// HMI/VISUs/Cryo-Routines/Cool-Down/VISU_HMI_COOL_DOWN
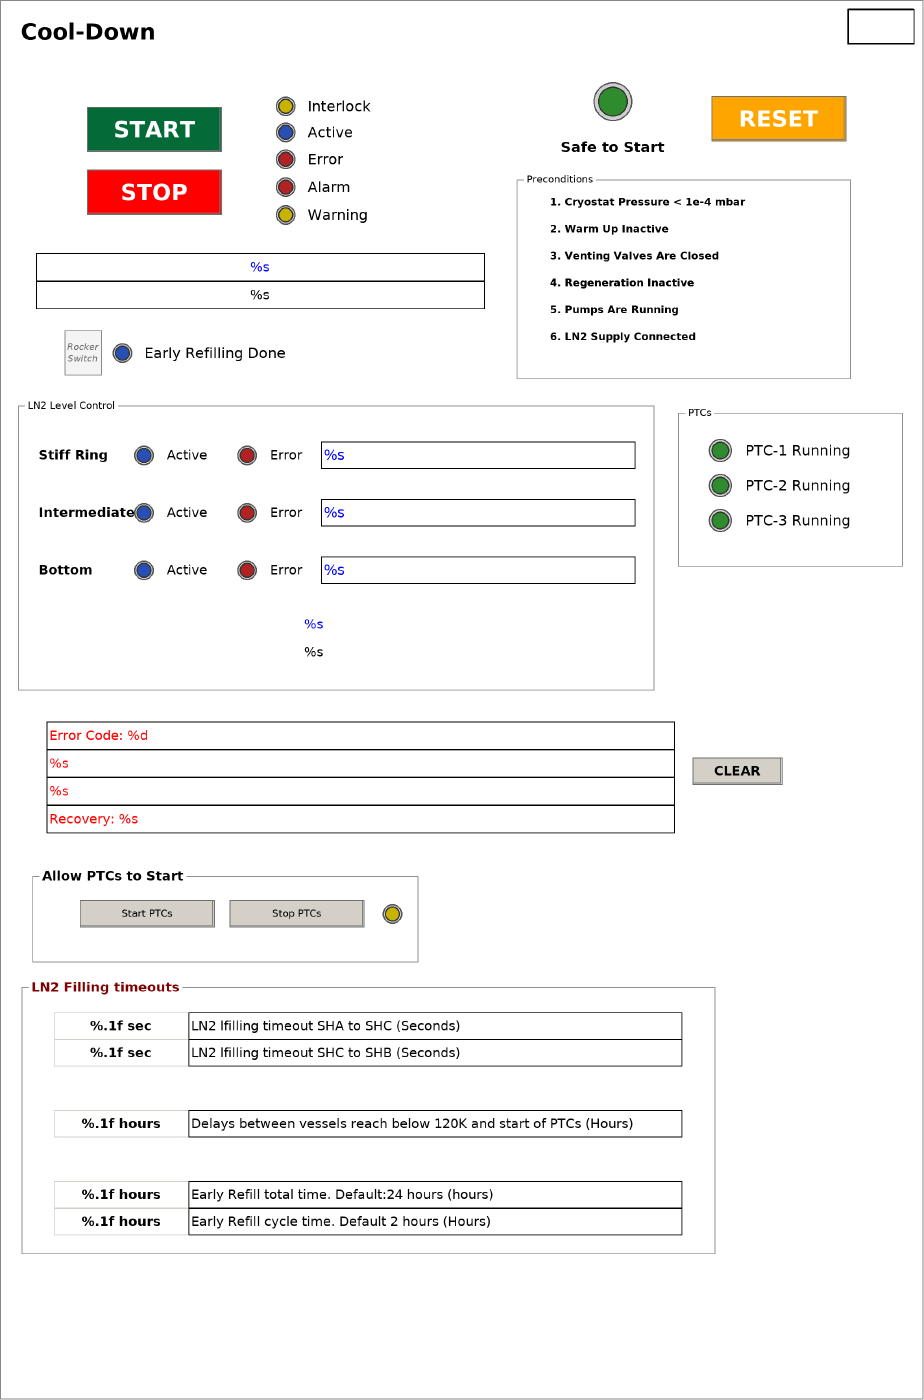
VISUALIZATION VISU_HMI_COOL_DOWN  // 1030x1560
VAR_IN_OUT
	m_instance : FB_METIS_CRYO_COOL_DOWN;
	m_Cry_Instance:	FB_METIS_CRYO_CTRL;	
END_VAR
    Label (20,20 163x30), "Cool-Down"
    Rectangle (40,282 500x31), "%s", text variable: m_instance.stat.sState
    Group (97,103 334x152)
        Group (0,16 150x120)
            Button (0,70 150x50), "STOP"
                OnMouseClick: execute { m_instance.ctrl.bEnable := FALSE; }
            Button (0,0 150x50), "START", input disabled if: NOT m_instance.stat.bPreConditionsMet
                OnMouseClick: execute { m_instance.ctrl.bEnable := TRUE; m_Cry_Instance.ctrl.bEnable_Cool_Down := TRUE; }
        Group (209,0 125x152)
            Label (34,29 91x31), "Active"
            Lamp1 (0,32 25x25), variable: m_instance.stat.bActive, style: Lamp-Lamp1-Blue
            Label (34,59 90x31), "Error"
            Lamp1 (0,62 25x25), variable: m_instance.stat.bError, style: Lamp-Lamp1-Red
            Lamp1 (0,3 25x25), variable: m_instance.interlocks.bInterlock_CoolDown, style: Lamp-Lamp1-Yellow
            Label (34,0 91x31), "Interlock"
            Label (34,90 90x31), "Alarm"
            Lamp1 (0,93 25x25), variable: m_instance.stat.bAlarm, style: Lamp-Lamp1-Red
            Label (34,121 90x31), "Warning"
            Lamp1 (0,124 25x25), variable: m_instance.stat.bWarning, style: Lamp-Lamp1-Yellow
    Lamp1 (658,88 50x50), variable: NOT m_instance.interlocks.bInterlock_CoolDown AND m_instance.stat.bPreConditionsMet, style: Lamp-Lamp1-Green
    Rectangle (608,149 150x30), "Safe to Start"
    GroupBox (576,192 372x230), "Preconditions"
        Rectangle (34,78 300x30), "3. Venting Valves Are Closed", colour toggle: m_instance.in_Cryo_Stat.bVentingValvesAreClosed
        Rectangle (34,108 300x30), "4. Regeneration Inactive", colour toggle: NOT m_instance.in_Cryo_Stat.bRegenerationActive
        Rectangle (34,138 300x30), "5. Pumps Are Running", colour toggle: m_instance.in_Cryo_Stat.bPumpsAreRunning
        Rectangle (34,168 300x30), "6. LN2 Supply Connected", colour toggle: m_instance.bESO_LN2_Supply
    Rectangle (610,300 300x30), "4. Regeneration Inactive", colour toggle: NOT m_instance.in_Cryo_Stat.bRegenerationActive
    Rectangle (610,210 300x30), "1. Cryostat Pressure < 1e-4 mbar", colour toggle: m_instance.in_Cryo_Stat.bInVacuum
    Rectangle (610,240 300x30), "2. Warm Up Inactive", colour toggle: NOT m_instance.in_Cryo_Stat.bWarmUpActive
    Button (793,107 150x50), "RESET", invisible if: NOT m_instance.stat.bError
        OnMouseClick: execute { m_instance.ctrl.bReset := TRUE; }
    Rectangle (52,835 700x31), "%s", text variable: m_instance.stat.Error.sMessage
    Rectangle (52,804 700x31), "Error Code: %d", text variable: m_instance.stat.Error.nCode
    GroupBox (756,452 250x179), "PTCs"
        Group (32,35 187x108)
            Group (0,0 187x30)
                Lamp1 (0,0 30x30), tooltip "If ON, compressor is running", variable: m_Instance.ptc[1].stat.bSystemOn, style: Lamp-Lamp1-Green
                Rectangle (40,0 147x30), "PTC-1 Running", tooltip "Compressor is running"
            Group (0,39 187x30)
                Lamp1 (0,0 30x30), tooltip "If ON, compressor is running", variable: m_Instance.ptc[2].stat.bSystemOn, style: Lamp-Lamp1-Green
                Rectangle (40,0 147x30), "PTC-2 Running", tooltip "Compressor is running"
            Group (0,78 187x30)
                Lamp1 (0,0 30x30), tooltip "If ON, compressor is running", variable: m_Instance.ptc[3].stat.bSystemOn, style: Lamp-Lamp1-Green
                Rectangle (40,0 147x30), "PTC-3 Running", tooltip "Compressor is running"
    GroupBox (20,444 709x325), "LN2 Level Control"
        Group (20,48 668x158)
            Group (0,64 668x30)
                Group (0,0 318x30)
                    Lamp1 (108,3 25x25), tooltip "pump speed > 0 rpm", variable: m_instance.lc_ln2_level_ctrl[2].bActive, style: Lamp-Lamp1-Blue
                    Label (143,0 60x30), "Active"
                    Lamp1 (223,3 25x25), tooltip "pump speed > 0 rpm", variable: m_instance.lc_ln2_level_ctrl[2].bError, style: Lamp-Lamp1-Red
                    Label (258,0 60x30), "Error"
                    Label (0,0 100x30), "Intermediate"
                Rectangle (318,0 350x30), "%s", text variable: m_instance.lc_ln2_level_ctrl[2].LN2_Level.stat.sStatus
            Group (0,128 668x30)
                Group (0,0 318x30)
                    Lamp1 (108,3 25x25), tooltip "pump speed > 0 rpm", variable: m_instance.lc_ln2_level_ctrl[3].bActive, style: Lamp-Lamp1-Blue
                    Label (143,0 60x30), "Active"
                    Lamp1 (223,3 25x25), tooltip "pump speed > 0 rpm", variable: m_instance.lc_ln2_level_ctrl[3].bError, style: Lamp-Lamp1-Red
                    Label (258,0 60x30), "Error"
                    Label (0,0 100x30), "Bottom"
                Rectangle (318,0 350x30), "%s", text variable: m_instance.lc_ln2_level_ctrl[3].LN2_Level.stat.sStatus
            Group (0,0 668x30)
                Group (0,0 318x30)
                    Lamp1 (108,3 25x25), tooltip "pump speed > 0 rpm", variable: m_instance.lc_ln2_level_ctrl[1].bActive, style: Lamp-Lamp1-Blue
                    Label (143,0 60x30), "Active"
                    Lamp1 (223,3 25x25), tooltip "pump speed > 0 rpm", variable: m_instance.lc_ln2_level_ctrl[1].bError, style: Lamp-Lamp1-Red
                    Label (258,0 60x30), "Error"
                    Label (0,0 100x30), "Stiff Ring"
                Rectangle (318,0 350x30), "%s", text variable: m_instance.lc_ln2_level_ctrl[1].LN2_Level.stat.sStatus
        Rectangle (80,236 500x31), "%s", text variable: m_instance.stat.sEarlyFillState
        Rectangle (80,267 500x31), "%s", text variable: m_instance.stat.sEarlyFillSubState
    Rectangle (52,866 700x31), "%s", text variable: m_instance.stat.sErrorMessage
    Rectangle (52,897 700x31), "Recovery: %s", text variable: m_instance.stat.sRecoverySuggestion
    Frame (945,10 75x40)
        shows VISU_HMI_SUBSYSTEM_BUTTON(m_Hmi := PRG_HMI.fbBackButton)
        OnMouseClick: execute { PRG_HMI.eActiveTab := PRG_HMI.ePreviousTab; }
    Rectangle (40,313 500x31), "%s", text variable: m_instance.stat.sSubState
    GroupBox (36,968 430x104), "Allow PTCs to Start"
        Button (53,35 150x30), "Start PTCs", tooltip "Allow PTCs to start"
            OnMouseClick: execute { m_instance.bAllowPTCsStart := TRUE; }
        Button (220,35 150x30), "Stop PTCs", tooltip "Do not allow PTCs to start"
            OnMouseClick: execute { m_instance.bAllowPTCsStart := FALSE; }
        Lamp1 (389,38 25x25), variable: m_instance.bAllowPTCsStart, style: Lamp-Lamp1-Yellow
    GroupBox (24,1092 773x305), "LN2 Filling timeouts"
        Group (36,36 700x248)
            Group (0,0 700x60)
                Group (0,0 700x30)
                    Textfield (0,0 150x30), "%.1f sec", tooltip "(Seconds) LN2 lfilling timeout SHA to SHC", text variable: m_instance.lrDelaySHC
                        OnMouseClick: write the text variable via Default
                    Rectangle (150,0 550x30), "LN2 lfilling timeout SHA to SHC (Seconds)", text variable: m_instance.lrDelaySHC
                Group (0,30 700x30)
                    Textfield (0,0 150x30), "%.1f sec", tooltip "(Seconds) LN2 lfilling timeout SHC to SHB", text variable: m_instance.lrDelaySHB
                        OnMouseClick: write the text variable via Default
                    Rectangle (150,0 550x30), "LN2 lfilling timeout SHC to SHB (Seconds)"
            Group (0,109 700x30)
                Textfield (0,0 150x30), "%.1f hours", tooltip "(Hours) delays between vessels reach below 120K and start of PTCs", text variable: m_instance.lrDelaySHCold
                    OnMouseClick: write the text variable via Default
                Rectangle (150,0 550x30), "Delays between vessels reach below 120K and start of PTCs (Hours)"
            Group (0,188 700x60)
                Group (0,0 700x30)
                    Textfield (0,0 150x30), "%.1f hours", tooltip "(Hours) Early Refill total time (24 hours)", text variable: m_instance.lrEarlyRefillTotal
                        OnMouseClick: write the text variable via Default
                    Rectangle (150,0 550x30), "Early Refill total time. Default:24 hours (hours)"
                Group (0,30 700x30)
                    Textfield (0,0 150x30), "%.1f hours", tooltip "(Hours) Early Refill cycle time.", text variable: m_instance.lrEarlyRefillCycle
                        OnMouseClick: write the text variable via Default
                    Rectangle (150,0 550x30), "Early Refill cycle time. Default 2 hours (Hours)"
    Group (72,368 253x50)
        RockerSwitch (0,0 41x50), variable: m_instance.bEarlyRefillDone, behaviour: TOGGLE, style: Switch-RockerSwitch-Blue
        Lamp1 (52,13 25x25), variable: m_instance.bEarlyRefillDone, style: Lamp-Lamp1-Blue
        Label (86,10 167x31), "Early Refilling Done"
    Button (772,844 100x30), "CLEAR", tooltip "Clears Error texts"
        OnMouseClick: execute {
            m_instance.stat.Error.nCode := 0;
            m_instance.stat.Error.sMessage:= '';
            m_instance.stat.sErrorMessage := '';
            m_instance.stat.sRecoverySuggestion := '';
        }
END_VISUALIZATION

// HMI/VISUs/Cryo-Routines/Evacuation/VISU_HMI_EVACUATION
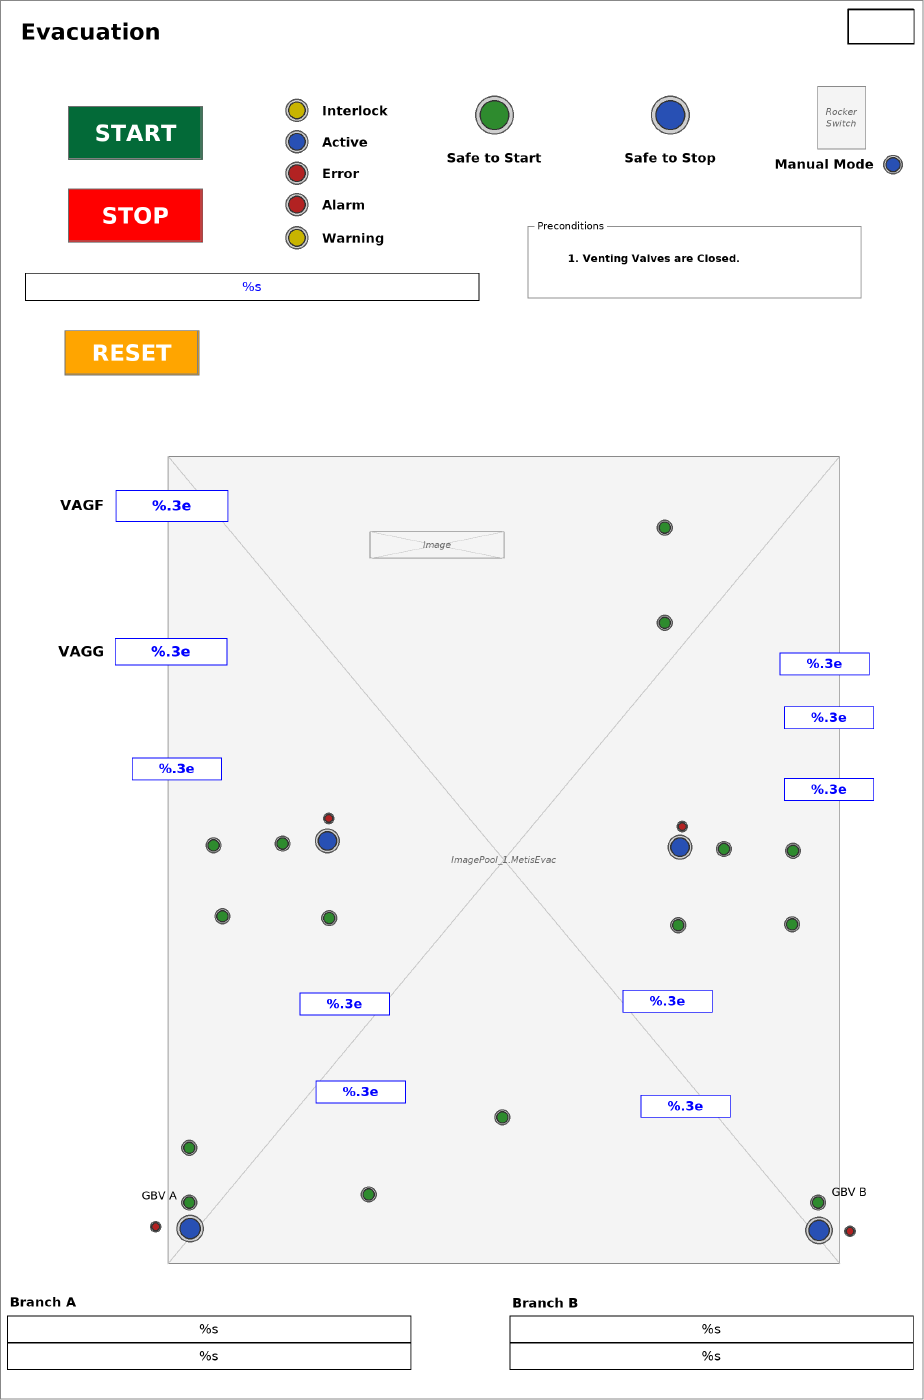
VISUALIZATION VISU_HMI_EVACUATION  // 1030x1560
    Label (20,20 163x30), "Evacuation"
    Frame (0,0 1030x1560)
        shows TEMPLATE_EVACUATION(m_Instance := MAIN.met_cryo_ctrl.met_evac, m_venting_instance := MAIN.met_cryo_ctrl.met_venting, m_cool_down_instance := MAIN.met_cryo_ctrl.met_cool_down)
    Frame (945,10 75x40)
        shows VISU_HMI_SUBSYSTEM_BUTTON(m_Hmi := PRG_HMI.fbBackButton)
        OnMouseClick: execute { PRG_HMI.eActiveTab := PRG_HMI.ePreviousTab; }
END_VISUALIZATION

// HMI/VISUs/Cryo-Routines/Power-Outage/VISU_HMI_POWER_OUTAGE
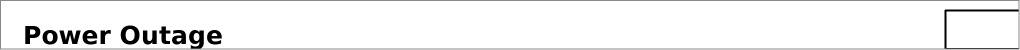
VISUALIZATION VISU_HMI_POWER_OUTAGE  // 1020x50
    Label (20,20 208x30), "Power Outage"
    Frame (945,10 75x40)
        shows VISU_HMI_SUBSYSTEM_BUTTON(m_Hmi := PRG_HMI.fbBackButton)
        OnMouseClick: execute { PRG_HMI.eActiveTab := PRG_HMI.ePreviousTab; }
END_VISUALIZATION

// HMI/VISUs/Cryo-Routines/Regeneration/VISU_HMI_REGENERATION
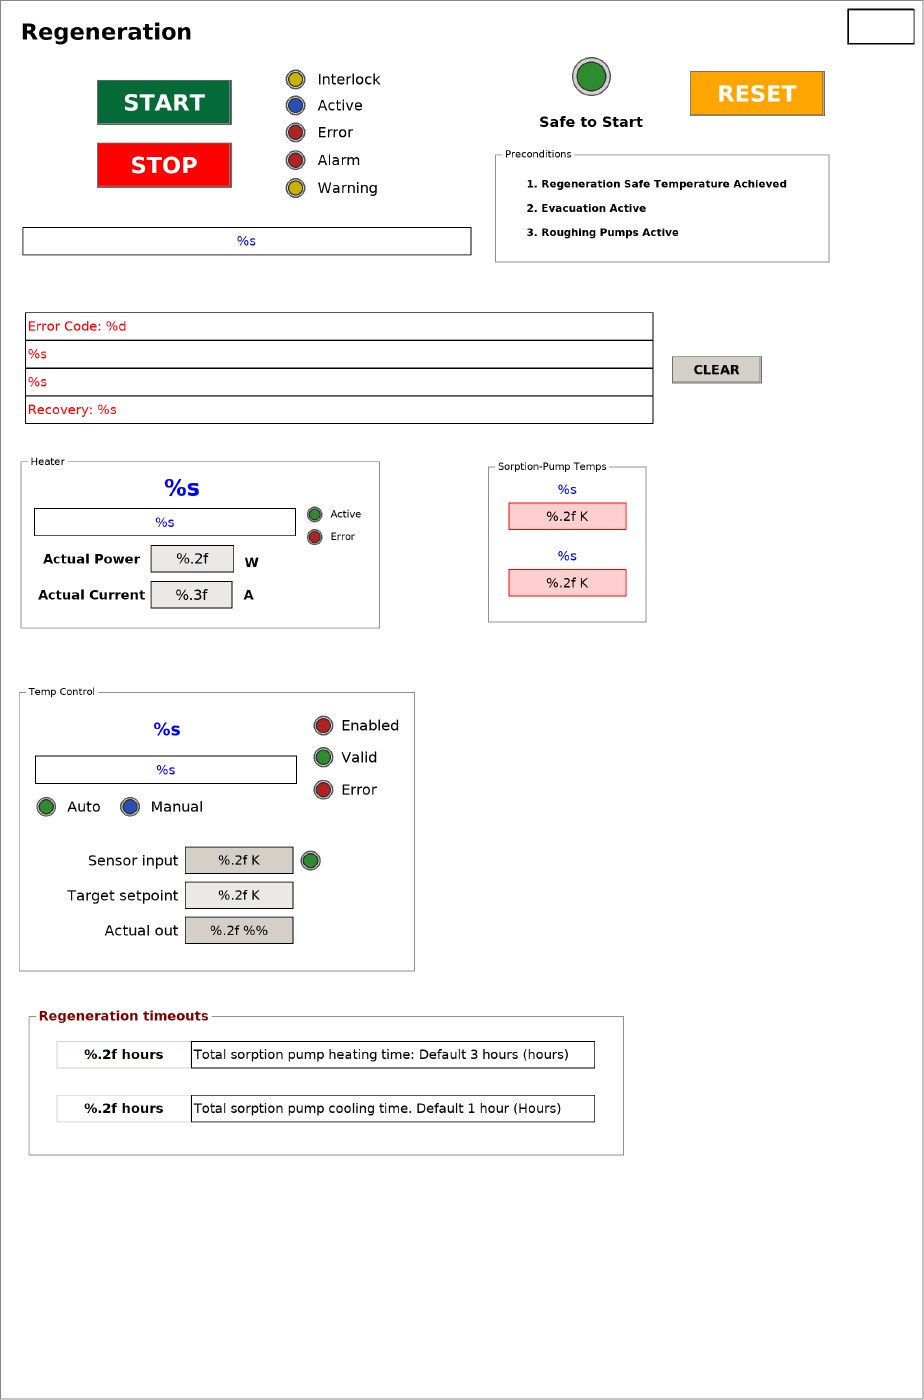
VISUALIZATION VISU_HMI_REGENERATION  // 1030x1560
VAR_IN_OUT
	//m_temp_instance : FB_METIS_TEMPERATURES;
	m_instance : FB_METIS_CRYO_REGENERATION;
	
END_VAR
    Label (20,20 194x30), "Regeneration"
    Frame (12,760 450x322)
        shows TEMPLATE_METIS_CTRL_TEMPERATURE_SIMPLIFIED(m_instance := MAIN.met_cryo_ctrl.met_tctrl.tc_cry_sp)
    Frame (16,504 407x196)
        shows TEMPLATE_METIS_HEATER_SIMPLIFIED(m_instance := MAIN.met_cryo_ctrl.met_heaters.h_cry_sp)
    Group (544,512 176x181)
        GroupBox (0,0 176x181), "Sorption-Pump Temps"
        Group (13,18 150x144)
            Frame (0,0 150x70)
                shows TEMPLATE_TEMP_SENSOR_VALUE_ONLY(m_instance := MAIN.met_cryo_ctrl.met_temp.t_cry_sp_1)
            Frame (0,74 150x70)
                shows TEMPLATE_TEMP_SENSOR_VALUE_ONLY(m_instance := MAIN.met_cryo_ctrl.met_temp.t_cry_sp_2)
    Rectangle (25,253 500x31), "%s", text variable: m_instance.stat.sState
    Group (108,73 334x152)
        Button (0,86 150x50), "STOP"
            OnMouseClick: execute { m_instance.ctrl.bEnable := FALSE; }
        Button (0,16 150x50), "START", input disabled if: m_instance.interlocks.bInterlock_Regeneration OR NOT m_instance.stat.bPreConditionsMet
            OnMouseClick: execute { m_instance.ctrl.bEnable := TRUE; }
        Group (209,0 125x152)
            Label (34,29 91x31), "Active"
            Lamp1 (0,32 25x25), variable: m_instance.stat.bActive, style: Lamp-Lamp1-Blue
            Label (34,59 90x31), "Error"
            Lamp1 (0,62 25x25), variable: m_instance.stat.bError, style: Lamp-Lamp1-Red
            Lamp1 (0,3 25x25), variable: m_instance.interlocks.bInterlock_Regeneration, style: Lamp-Lamp1-Yellow
            Label (34,0 91x31), "Interlock"
            Label (34,90 90x31), "Alarm"
            Lamp1 (0,93 25x25), variable: m_instance.stat.bAlarm, style: Lamp-Lamp1-Red
            Label (34,121 90x31), "Warning"
            Lamp1 (0,124 25x25), variable: m_instance.stat.bWarning, style: Lamp-Lamp1-Yellow
    Lamp1 (634,60 50x50), variable: NOT m_instance.interlocks.bInterlock_Regeneration, style: Lamp-Lamp1-Green
    Rectangle (584,121 150x30), "Safe to Start"
    GroupBox (552,164 372x128), "Preconditions"
        Rectangle (32,80 300x30), "3. Roughing Pumps Active", colour toggle: m_instance.in_Cryo_Stat.bRoughingPumpsAreRunning
    Rectangle (584,190 300x30), "1. Regeneration Safe Temperature Achieved", colour toggle: (m_instance.in_Cryo_Stat.lrLowestTempK >= m_instance.in_lrRegeneration_Safe_Temp)
    Rectangle (584,217 300x30), "2. Evacuation Active", colour toggle: m_instance.in_Cryo_Stat.bEvacuationActive
    Button (769,79 150x50), "RESET", invisible if: NOT m_instance.stat.bError
        OnMouseClick: execute { m_instance.ctrl.bReset := TRUE; }
    Frame (945,10 75x40)
        shows VISU_HMI_SUBSYSTEM_BUTTON(m_Hmi := PRG_HMI.fbBackButton)
        OnMouseClick: execute { PRG_HMI.eActiveTab := PRG_HMI.ePreviousTab; }
    Rectangle (28,379 700x31), "%s", text variable: m_instance.stat.Error.sMessage
    Rectangle (28,348 700x31), "Error Code: %d", text variable: m_instance.stat.Error.nCode
    Rectangle (28,410 700x31), "%s", text variable: m_instance.stat.sErrorMessage
    Rectangle (28,441 700x31), "Recovery: %s", text variable: m_instance.stat.sRecoverySuggestion
    GroupBox (32,1124 663x163), "Regeneration timeouts"
        Group (31,36 600x90)
            Group (0,0 600x30)
                Textfield (0,0 150x30), "%.2f hours", tooltip "(Hours) Total heating time", text variable: m_instance.lrHeatingTime
                    OnMouseClick: write the text variable via Default
                Rectangle (150,0 450x30), "Total sorption pump heating time: Default 3 hours (hours)"
            Group (0,60 600x30)
                Textfield (0,0 150x30), "%.2f hours", tooltip "(Hours) Total Cooling time", text variable: m_instance.lrCoolDownTime
                    OnMouseClick: write the text variable via Default
                Rectangle (150,0 450x30), "Total sorption pump cooling time. Default 1 hour (Hours)"
    Button (749,397 100x30), "CLEAR", tooltip "Clears Error texts"
        OnMouseClick: execute {
            m_instance.stat.Error.nCode := 0;
            m_instance.stat.Error.sMessage:= '';
            m_instance.stat.sErrorMessage := '';
            m_instance.stat.sRecoverySuggestion := '';
        }
END_VISUALIZATION

// HMI/VISUs/Cryo-Routines/Regeneration/VISU_REGENERATION_CTRL
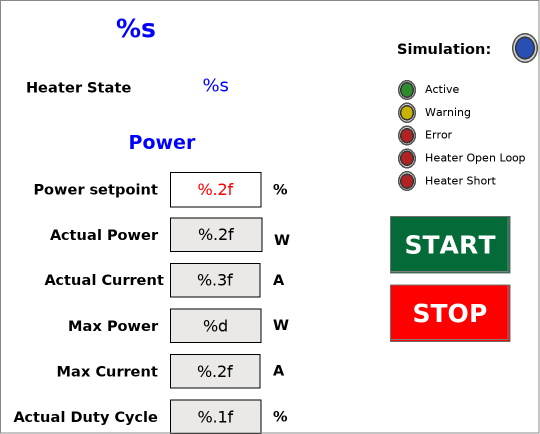
VISUALIZATION VISU_REGENERATION_CTRL  // 540x434
    Frame (0,0 540x434)
        shows TEMPLATE_HEATER_PWM_CTRL(m_instance := MAIN.met_cryo_ctrl.met_regeneration.h_sorption_pump_heater, m_bEnable := MAIN.met_cryo_ctrl.met_regeneration.h_sorption_pump_heater.ctrl.bEnable)
END_VISUALIZATION

// HMI/VISUs/Cryo-Routines/Regeneration/VISU_SORPTION_HEATER
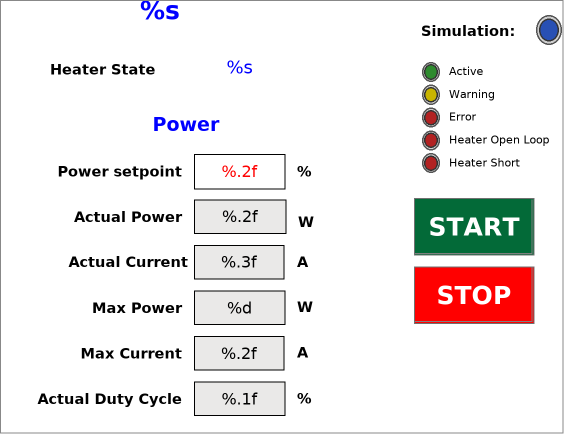
VISUALIZATION VISU_SORPTION_HEATER  // 564x434
    Frame (24,-18 540x434)
        shows TEMPLATE_HEATER_PWM_CTRL(m_instance := MAIN.met_cryo_ctrl.met_regeneration.h_sorption_pump_heater, m_bEnable := MAIN.met_cryo_ctrl.met_regeneration.h_sorption_pump_heater.ctrl.bEnable)
END_VISUALIZATION

// HMI/VISUs/Cryo-Routines/Regeneration/VISU_SORPTION_TEMP_VOTE
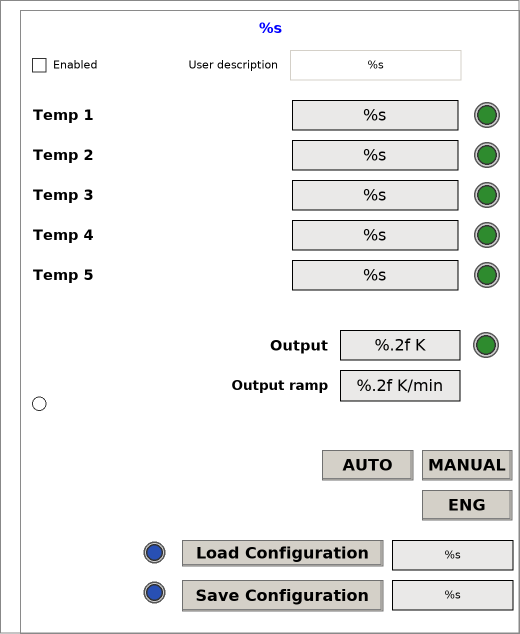
VISUALIZATION VISU_SORPTION_TEMP_VOTE  // 520x634
    Frame (20,10 500x624)
        shows TEMPLATE_TEMPERATURE_VOTE(m_Instance := MAIN.met_cryo_ctrl.met_regeneration.t_vote_tc_cry_sp, m_all_temperatures_array := MAIN.met_cryo_ctrl.met_temp)
END_VISUALIZATION

// HMI/VISUs/Cryo-Routines/Venting/VISU_HMI_VENTING
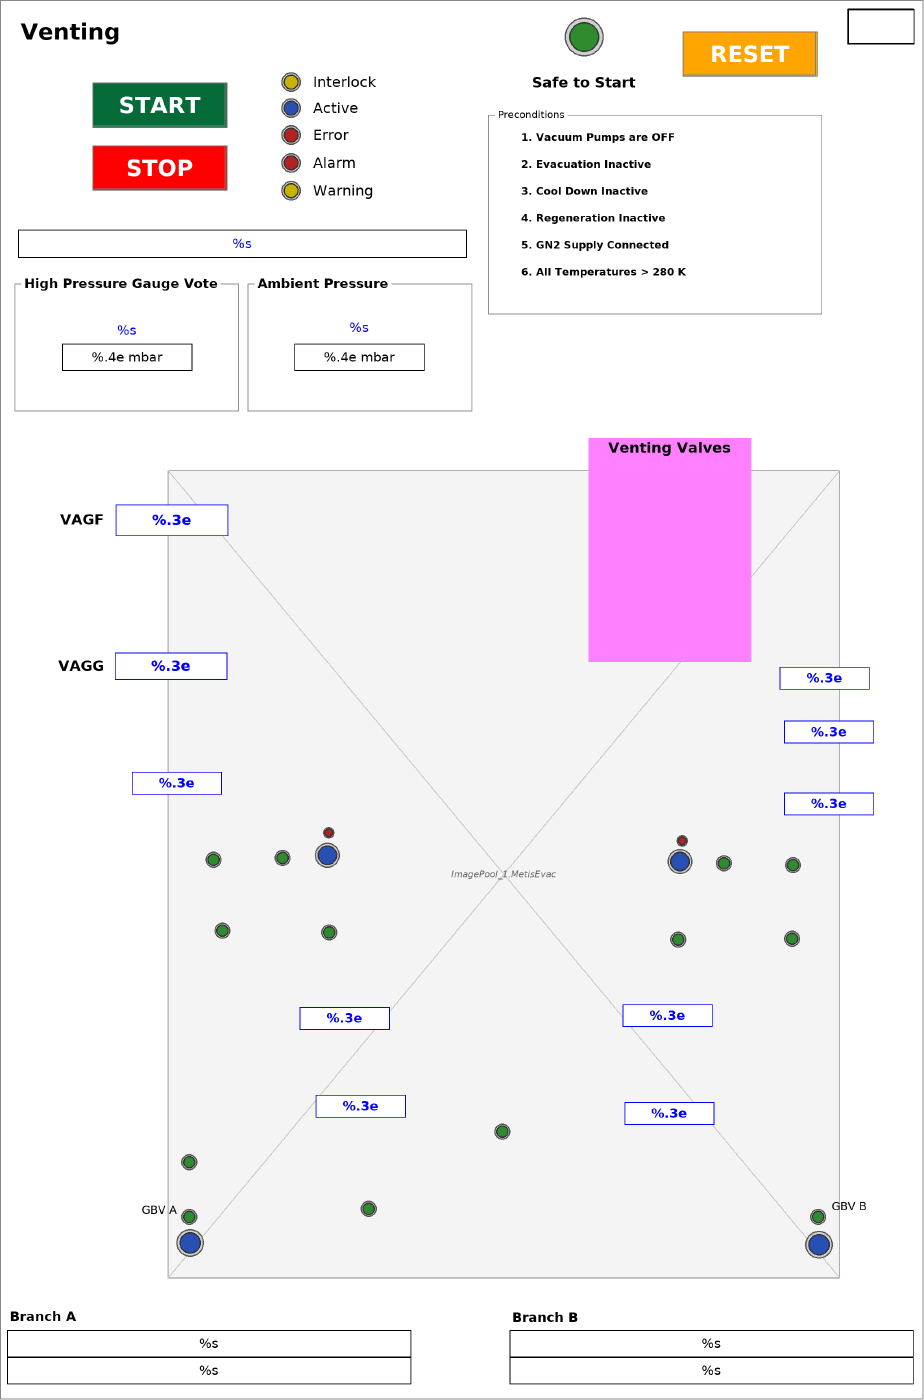
VISUALIZATION VISU_HMI_VENTING  // 1030x1560
VAR_IN_OUT
	m_Instance : FB_METIS_CRYO_VENTING;
	m_Cry_Instance:	FB_METIS_CRYO_CTRL;
END_VAR
    Image (187,524 749x900), image: ImagePool_1.MetisEvac
    Label (20,20 163x30), "Venting"
    Rectangle (20,256 500x31), "%s", text variable: m_instance.stat.sState
    Button (103,162 150x50), "STOP"
        OnMouseClick: execute { m_instance.ctrl.bEnable := FALSE; m_Cry_Instance.ctrl.bEnable_Venting := FALSE; }
    Button (103,92 150x50), "START", input disabled if: NOT m_instance.stat.bPreConditionsMet OR m_instance.interlocks.bInterlock_Venting
        OnMouseClick: execute { m_instance.ctrl.bEnable := TRUE; m_Cry_Instance.ctrl.bEnable_Venting := TRUE; }
    Label (346,105 91x31), "Active"
    Lamp1 (312,108 25x25), variable: m_instance.stat.bActive, style: Lamp-Lamp1-Blue
    Label (346,135 90x31), "Error"
    Lamp1 (312,138 25x25), variable: m_instance.stat.bError, style: Lamp-Lamp1-Red
    Lamp1 (312,79 25x25), variable: m_instance.interlocks.bInterlock_Venting, style: Lamp-Lamp1-Yellow
    Label (346,76 91x31), "Interlock"
    Label (346,166 90x31), "Alarm"
    Lamp1 (312,169 25x25), variable: m_instance.stat.bAlarm, style: Lamp-Lamp1-Red
    Label (346,197 90x31), "Warning"
    Lamp1 (312,200 25x25), variable: m_instance.stat.bWarning, style: Lamp-Lamp1-Yellow
    Lamp1 (626,16 50x50), variable: NOT m_instance.interlocks.bInterlock_Venting AND m_instance.stat.bPreConditionsMet, style: Lamp-Lamp1-Green
    Rectangle (576,77 150x30), "Safe to Start"
    GroupBox (544,120 372x230), "Preconditions"
        Rectangle (34,78 300x30), "3. Cool Down Inactive", colour toggle: NOT m_instance.in_Cryo_Stat.bCoolDownActive
        Rectangle (34,108 300x30), "4. Regeneration Inactive", colour toggle: NOT m_instance.in_Cryo_Stat.bRegenerationActive
        Rectangle (34,138 300x30), "5. GN2 Supply Connected", colour toggle: m_instance.in_Cryo_Stat.bGN2SupplyConnected
        Rectangle (34,168 300x30), "6. All Temperatures > 280 K", colour toggle: m_instance.in_Cryo_Stat.lrLowestTempK > 280.0
    Rectangle (578,138 300x30), "1. Vacuum Pumps are OFF", colour toggle: NOT m_instance.in_Cryo_Stat.bPumpsAreRunning
    Rectangle (578,168 300x30), "2. Evacuation Inactive", colour toggle: NOT m_instance.in_Cryo_Stat.bEvacuationActive
    Button (761,35 150x50), "RESET", invisible if: NOT m_instance.stat.bError
        OnMouseClick: execute { m_instance.ctrl.bReset := TRUE; }
    Frame (945,10 75x40)
        shows VISU_HMI_SUBSYSTEM_BUTTON(m_Hmi := PRG_HMI.fbBackButton)
        OnMouseClick: execute { PRG_HMI.eActiveTab := PRG_HMI.ePreviousTab; }
    GroupBox (276,308 250x150), "Ambient Pressure"
        Frame (50,40 150x70)
            shows TEMPLATE_AMBIENT_PRESSURE_READING(m_instance := MAIN.met_cryo_ctrl.sensor_AMB_PRESS)
    GroupBox (16,308 250x150), "High Pressure Gauge Vote", tooltip "Pressure vote of HPG1 and HPG2"
        Group (53,45 145x60)
            Rectangle (0,30 145x30), "%.4e mbar", tooltip "Pressure in mbar", text variable: m_instance.HPG.stat.lrPressure
            Rectangle (0,0 145x30), "%s", text variable: m_instance.HPG.in_sName
    Rectangle (8,1482 450x30), "%s", text variable: m_Cry_Instance.met_evac.evac_branch_a.stat.sErrorText
    Rectangle (8,1512 450x30), "%s", text variable: m_Cry_Instance.met_evac.evac_branch_a.stat.sStatus
    Rectangle (8,1452 100x30), "Branch A"
    Rectangle (568,1482 450x30), "%s", text variable: m_Cry_Instance.met_evac.evac_branch_b.stat.sErrorText
    Rectangle (568,1512 450x30), "%s", text variable: m_Cry_Instance.met_evac.evac_branch_b.stat.sStatus
    Rectangle (568,1453 100x30), "Branch B"
    Rectangle (334,1122 100x25), "%.3e", text variable: m_Cry_Instance.met_evac.evac_branch_a.VAG1.stat.lrPressure
    Rectangle (147,860 100x25), "%.3e", text variable: m_Cry_Instance.met_evac.evac_branch_a.VAG2.stat.lrPressure
    Lamp1 (194,1367 36x36), variable: m_Cry_Instance.met_evac.evac_branch_a.rp.stat.bReady, style: Lamp-Lamp1-Blue
    Lamp1 (349,937 32x32), tooltip "If ON, TMP pump is at its nominal speed, i.e. Ready.", variable: m_Cry_Instance.met_evac.evac_branch_a.tp.stat.bReady, style: Lamp-Lamp1-Blue
    Lamp1 (238,1027 20x20), variable: m_Cry_Instance.met_evac.evac_branch_a.PVV1.stat.bActON, style: Lamp-Lamp1-Green
    Lamp1 (357,1029 20x20), variable: m_Cry_Instance.met_evac.evac_branch_a.PVV2.stat.bActON, style: Lamp-Lamp1-Green
    Lamp1 (228,948 20x20), variable: m_Cry_Instance.met_evac.evac_branch_a.PVV3.stat.bActON, style: Lamp-Lamp1-Green
    Lamp1 (305,946 20x20), variable: m_Cry_Instance.met_evac.evac_branch_a.PVV4.stat.bActON, style: Lamp-Lamp1-Green
    Lamp1 (201,1346 20x20), variable: m_Cry_Instance.met_evac.evac_branch_a.GBV.stat.bActON, style: Lamp-Lamp1-Green
    Lamp1 (359,921 15x14), tooltip "If ON, TMP pump is still spinning.", variable: m_Cry_Instance.met_evac.evac_branch_a.tp.stat.bSpeed100, style: Lamp-Lamp1-Red
    Rectangle (352,1220 100x25), "%.3e", text variable: m_Cry_Instance.met_evac.evac_branch_a.VAG3.stat.lrPressure
    Lamp1 (742,944 32x32), tooltip "If ON, TMP pump is at its nominal speed, i.e. Ready.", variable: m_Cry_Instance.met_evac.evac_branch_b.tp.stat.bReady, style: Lamp-Lamp1-Blue
    Lamp1 (753,930 15x14), tooltip "If ON, TMP pump is still spinning.", variable: m_Cry_Instance.met_evac.evac_branch_b.tp.stat.bSpeed100, style: Lamp-Lamp1-Red
    Lamp1 (797,952 20x20), variable: m_Cry_Instance.met_evac.evac_branch_b.PVV4.stat.bActON, style: Lamp-Lamp1-Green
    Lamp1 (874,954 20x20), variable: m_Cry_Instance.met_evac.evac_branch_b.PVV3.stat.bActON, style: Lamp-Lamp1-Green
    Lamp1 (746,1037 20x20), variable: m_Cry_Instance.met_evac.evac_branch_b.PVV2.stat.bActON, style: Lamp-Lamp1-Green
    Lamp1 (873,1036 20x20), variable: m_Cry_Instance.met_evac.evac_branch_b.PVV1.stat.bActON, style: Lamp-Lamp1-Green
    Lamp1 (895,1369 36x36), variable: m_Cry_Instance.met_evac.evac_branch_b.rp.stat.bReady, style: Lamp-Lamp1-Blue
    Lamp1 (902,1346 20x20), variable: m_Cry_Instance.met_evac.evac_branch_b.GBV.stat.bActON, style: Lamp-Lamp1-Green
    Rectangle (696,1228 100x25), "%.3e", text variable: m_Cry_Instance.met_evac.evac_branch_b.VAG3.stat.lrPressure
    Rectangle (874,883 100x25), "%.3e", text variable: m_Cry_Instance.met_evac.evac_branch_b.VAG2.stat.lrPressure
    Rectangle (694,1119 100x25), "%.3e", text variable: m_Cry_Instance.met_evac.evac_branch_b.VAG1.stat.lrPressure
    Lamp1 (728,592 25x25), variable: m_Instance.N2V_1.stat.bActON, style: Lamp-Lamp1-Green
    Lamp1 (728,696 25x25), variable: m_Instance.N2V_2.stat.bActON, style: Lamp-Lamp1-Green
    Lamp1 (201,1285 20x20), variable: m_Cry_Instance.met_cool_down.PVV_P1.stat.bActON, style: Lamp-Lamp1-Green
    Lamp1 (401,1337 20x20), variable: m_Cry_Instance.met_cool_down.PVV_P3.stat.bActON, style: Lamp-Lamp1-Green
    Lamp1 (550,1251 20x20), variable: m_Cry_Instance.met_cool_down.PVV_P2.stat.bActON, style: Lamp-Lamp1-Green
    Rectangle (150,1333 55x30), "GBV A"
    Rectangle (919,1329 55x30), "GBV B"
    Rectangle (129,562 125x35), "%.3e", text variable: m_Cry_Instance.met_evac.VAGF.stat.lrPressure
    Rectangle (54,564 75x30), "VAGF"
    Rectangle (128,727 125x30), "%.3e", text variable: m_Cry_Instance.met_evac.VAGG.stat.lrPressure
    Rectangle (53,727 75x30), "VAGG"
    Rectangle (869,743 100x25), "%.3e", text variable: m_Instance.sensor_HPG1.stat.lrPressure
    Rectangle (874,803 100x25), "%.3e", text variable: m_Instance.sensor_HPG2.stat.lrPressure
    Rectangle (656,488 181x249), "Venting Valves"
END_VISUALIZATION

// HMI/VISUs/Cryo-Routines/Warm-Up/VISU_HMI_WARM_UP
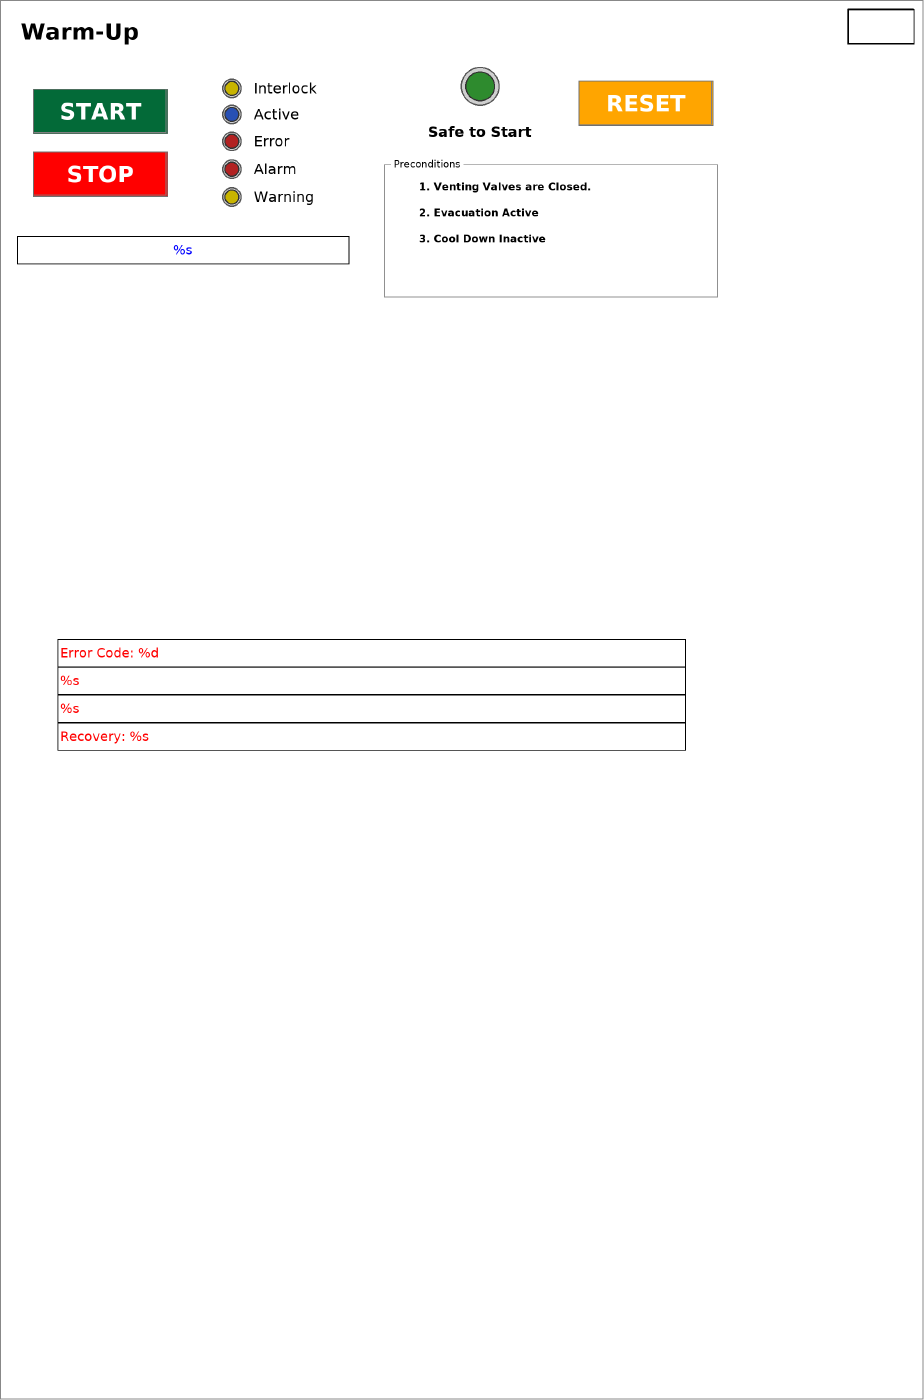
VISUALIZATION VISU_HMI_WARM_UP  // 1030x1560
VAR_IN_OUT
	m_instance : FB_METIS_CRYO_WARM_UP;
	m_Cry_Instance:	FB_METIS_CRYO_CTRL;
END_VAR
    Label (20,20 163x30), "Warm-Up"
    Rectangle (19,263 370x31), "%s", text variable: m_instance.stat.sState
    Button (37,169 150x50), "STOP"
        OnMouseClick: execute { m_instance.ctrl.bEnable := FALSE; }
    Button (37,99 150x50), "START", input disabled if: NOT m_instance.stat.bPreConditionsMet OR m_instance.interlocks.bInterlock_WarmUp
        OnMouseClick: execute { m_instance.ctrl.bEnable := TRUE; m_Cry_Instance.ctrl.bEnable_Warm_Up := TRUE; }
    Label (280,112 91x31), "Active"
    Lamp1 (246,115 25x25), variable: m_instance.stat.bActive, style: Lamp-Lamp1-Blue
    Label (280,142 90x31), "Error"
    Lamp1 (246,145 25x25), variable: m_instance.stat.bError, style: Lamp-Lamp1-Red
    Lamp1 (246,86 25x25), variable: m_instance.interlocks.bInterlock_WarmUp, style: Lamp-Lamp1-Yellow
    Label (280,83 91x31), "Interlock"
    Label (280,173 90x31), "Alarm"
    Lamp1 (246,176 25x25), variable: m_instance.stat.bAlarm, style: Lamp-Lamp1-Red
    Label (280,204 90x31), "Warning"
    Lamp1 (246,207 25x25), variable: m_instance.stat.bWarning, style: Lamp-Lamp1-Yellow
    Lamp1 (510,71 50x50), variable: NOT m_instance.interlocks.bInterlock_Regeneration, style: Lamp-Lamp1-Green
    Rectangle (460,132 150x30), "Safe to Start"
    GroupBox (428,175 372x156), "Preconditions"
        Rectangle (36,76 300x30), "3. Cool Down Inactive", colour toggle: NOT m_instance.in_Cryo_Stat.bCoolDownActive
    Rectangle (464,193 300x30), "1. Venting Valves are Closed.", colour toggle: m_instance.in_Cryo_Stat.bVentingValvesAreClosed
    Rectangle (464,222 300x30), "2. Evacuation Active", colour toggle: m_instance.in_Cryo_Stat.bEvacuationActive
    Button (645,90 150x50), "RESET", invisible if: NOT m_instance.stat.bError
        OnMouseClick: execute { m_instance.ctrl.bReset := TRUE; }
    Rectangle (64,743 700x31), "%s", text variable: m_instance.stat.Error.sMessage
    Rectangle (64,712 700x31), "Error Code: %d", text variable: m_instance.stat.Error.nCode
    Rectangle (64,774 700x31), "%s", text variable: m_instance.stat.sErrorMessage
    Rectangle (64,805 700x31), "Recovery: %s", text variable: m_instance.stat.sRecoverySuggestion
    Frame (945,10 75x40)
        shows VISU_HMI_SUBSYSTEM_BUTTON(m_Hmi := PRG_HMI.fbBackButton)
        OnMouseClick: execute { PRG_HMI.eActiveTab := PRG_HMI.ePreviousTab; }
END_VISUALIZATION

// HMI/VISUs/Events/VISU_HMI_EVENTS
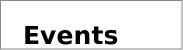
VISUALIZATION VISU_HMI_EVENTS  // 183x50
    Label (20,20 163x30), "Events"
END_VISUALIZATION

// HMI/VISUs/GUIs/GUI_LN2_LEVEL_CTRL
VISUALIZATION GUI_LN2_LEVEL_CTRL  // 2x2
END_VISUALIZATION

// HMI/VISUs/GUIs/GUI_MANUAL_CONTROL
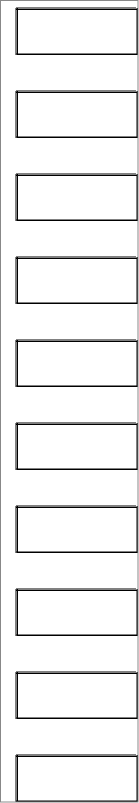
VISUALIZATION GUI_MANUAL_CONTROL  // 139x803
    Frame (16,672 123x48)
        shows VISU_HMI_SUBSYSTEM_BUTTON(m_Hmi := PRG_HMI.fbValvesButton)
        OnMouseClick: execute { PRG_HMI.eActiveTab := E_HMI_TABS.VALVES; }
    Frame (16,8 123x48)
        shows VISU_HMI_SUBSYSTEM_BUTTON(m_Hmi := PRG_HMI.fbCabinetsButton)
        OnMouseClick: execute { PRG_HMI.eActiveTab := E_HMI_TABS.CABINETS; }
    Frame (16,91 123x48)
        shows VISU_HMI_SUBSYSTEM_BUTTON(m_Hmi := PRG_HMI.fbControlUnitsButton)
        OnMouseClick: execute { PRG_HMI.eActiveTab := E_HMI_TABS.CONTROL_UNITS; }
    Frame (16,174 123x48)
        shows VISU_HMI_SUBSYSTEM_BUTTON(m_Hmi := PRG_HMI.fbCoolersButton)
        OnMouseClick: execute { PRG_HMI.eActiveTab := E_HMI_TABS.COOLERS; }
    Frame (16,257 123x48)
        shows VISU_HMI_SUBSYSTEM_BUTTON(m_Hmi := PRG_HMI.fbDetectorsButton)
        OnMouseClick: execute { PRG_HMI.eActiveTab := E_HMI_TABS.DETECTORS; }
    Frame (16,340 123x48)
        shows VISU_HMI_SUBSYSTEM_BUTTON(m_Hmi := PRG_HMI.fbHeatersButton)
        OnMouseClick: execute { PRG_HMI.eActiveTab := E_HMI_TABS.HEATERS; }
    Frame (16,506 123x48)
        shows VISU_HMI_SUBSYSTEM_BUTTON(m_Hmi := PRG_HMI.fbPressuresButton)
        OnMouseClick: execute { PRG_HMI.eActiveTab := E_HMI_TABS.PRESSURES; }
    Frame (16,589 123x48)
        shows VISU_HMI_SUBSYSTEM_BUTTON(m_Hmi := PRG_HMI.fbTemperaturesButton)
        OnMouseClick: execute { PRG_HMI.eActiveTab := E_HMI_TABS.TEMPERATURES; }
    Frame (16,423 123x48)
        shows VISU_HMI_SUBSYSTEM_BUTTON(m_Hmi := PRG_HMI.fbPumpsButton)
        OnMouseClick: execute { PRG_HMI.eActiveTab := E_HMI_TABS.PUMPS; }
    Frame (16,755 123x48)
        shows VISU_HMI_SUBSYSTEM_BUTTON(m_Hmi := PRG_HMI.fbControlLoopsButton)
        OnMouseClick: execute { PRG_HMI.eActiveTab := E_HMI_TABS.CONTROL_LOOPS; }
END_VISUALIZATION

// HMI/VISUs/GUIs/GUI_METIS_EVACUATION
VISUALIZATION GUI_METIS_EVACUATION  // 1500x950
END_VISUALIZATION

// HMI/VISUs/GUIs/VISU_HMI_FUSE_HMI
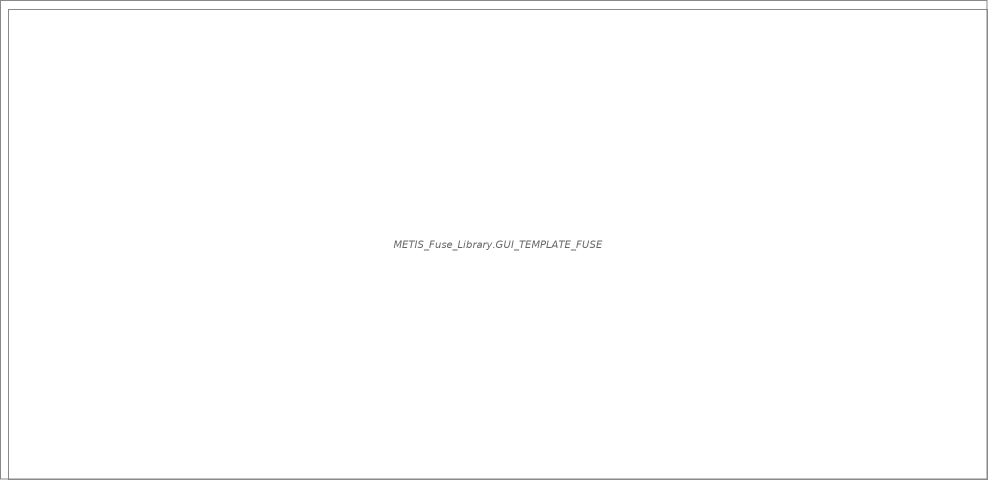
VISUALIZATION VISU_HMI_FUSE_HMI  // 988x480
    Frame (8,9 980x471)
        shows METIS_Fuse_Library.GUI_TEMPLATE_FUSE(m_Instance := MAIN.met_cryo_ctrl.fuseHMI)
END_VISUALIZATION

// HMI/VISUs/Home/VISU_HMI_HOME
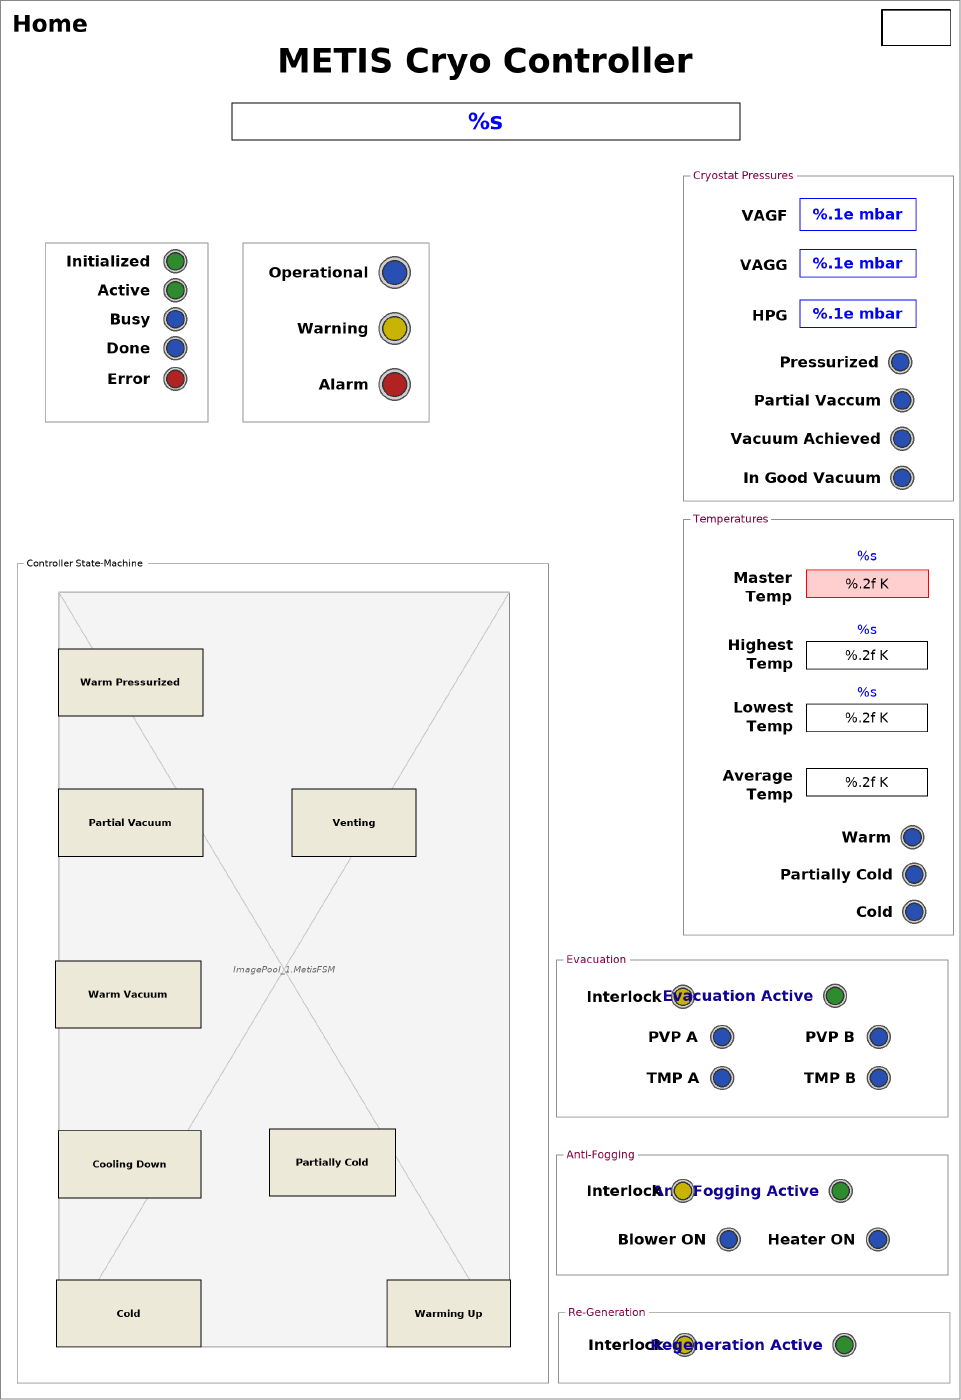
VISUALIZATION VISU_HMI_HOME  // 1030x1500
VAR_IN_OUT
	m_instance : FB_METIS_CRYO_CTRL;
END_VAR
    GroupBox (596,1229 420x137), "Anti-Fogging"
        Rectangle (10,20 400x105), colour toggle: m_instance.stat.bAntiFoggingActive
        Group (204,84 156x30)
            Lamp1 (126,0 30x30), tooltip "If ON, TMP pump is at its nominal speed, i.e. Ready.", variable: m_Instance.met_heaters.h_cry_wi.stat.bActive, style: Lamp-Lamp1-Blue
            Rectangle (0,0 120x30), "Heater ON"
        Group (44,84 156x30)
            Lamp1 (126,0 30x30), variable: m_Instance.met_anti_fogging.dryair_blow_valve.stat.bActive, style: Lamp-Lamp1-Blue
            Rectangle (0,0 120x30), "Blower ON"
        Group (101,32 219x30)
            Lamp1 (189,0 30x30), variable: m_instance.stat.bAntiFoggingActive, invisible if: NOT m_instance.stat.bAntiFoggingActive, style: Lamp-Lamp1-Green
            Rectangle (0,0 184x30), "Anti-Fogging Active", invisible if: NOT m_instance.stat.bAntiFoggingActive
        Group (16,32 135x30), invisible if: m_instance.stat.bAntiFoggingActive
            Lamp1 (105,0 30x30), variable: NOT m_instance.ctrl.bSafe_Anti_Fogging, style: Lamp-Lamp1-Yellow
            Rectangle (0,0 100x30), "Interlock"
    GroupBox (260,252 200x200)
        Group (18,20 165x160)
            Group (0,60 165x40)
                Rectangle (0,5 120x30), "Warning"
                Lamp1 (125,0 40x40), variable: m_instance.stat.bWarning, style: Lamp-Lamp1-Yellow
            Group (0,120 165x40)
                Lamp1 (125,0 40x40), variable: m_instance.stat.bAlarm, style: Lamp-Lamp1-Red
                Rectangle (0,5 120x30), "Alarm"
            Group (0,0 165x40)
                Rectangle (0,5 120x30), "Operational"
                Lamp1 (125,0 40x40), tooltip "System is ready for operations", variable: m_instance.stat.bOP, style: Lamp-Lamp1-Blue
    GroupBox (598,1398 420x84), "Re-Generation"
        Rectangle (10,16 400x53), colour toggle: m_instance.stat.bRegenerationActive
        Group (16,28 135x30), invisible if: m_instance.stat.bRegenerationActive
            Lamp1 (105,0 30x30), variable: NOT m_instance.ctrl.bSafe_Regeneration, style: Lamp-Lamp1-Yellow
            Rectangle (0,0 100x30), "Interlock"
        Group (98,28 224x30), invisible if: NOT m_instance.stat.bRegenerationActive
            Lamp1 (194,0 30x30), variable: m_instance.stat.bRegenerationActive, invisible if: NOT m_instance.stat.bRegenerationActive, style: Lamp-Lamp1-Green
            Rectangle (0,0 189x30), "Regeneration Active", invisible if: NOT m_instance.stat.bRegenerationActive
    GroupBox (732,548 290x454), "Temperatures"
        Group (17,32 256x412)
            Group (0,0 256x282)
                Group (0,0 255x70)
                    Frame (105,0 150x70)
                        shows TEMPLATE_TEMP_SENSOR_VALUE_ONLY(m_instance := MAIN.met_cryo_ctrl.met_temp.t_master)
                    Rectangle (0,28 103x42), "Master Temp"
                Group (1,79 255x63)
                    Rectangle (0,21 103x42), "Highest Temp"
                    Group (104,0 151x58)
                        Rectangle (0,0 151x31), "%s", text variable: m_instance.stat.sHighestTempName
                        Rectangle (10,28 130x30), "%.2f K", tooltip "Highest of all temperatures", text variable: m_instance.stat.lrHighestTempK
                Group (1,146 255x63)
                    Rectangle (0,21 103x42), "Lowest Temp"
                    Group (104,0 151x58)
                        Rectangle (0,0 151x31), "%s", text variable: m_instance.stat.sLowestTempName
                        Rectangle (10,28 130x30), "%.2f K", tooltip "Lowest of all temperatures", text variable: m_instance.stat.lrLowestTempK
                Group (1,240 244x42)
                    Rectangle (0,0 103x42), "Average Temp"
                    Rectangle (114,3 130x30), "%.2f K", tooltip "Average of all temperatures", text variable: m_instance.stat.lrAverageOfAllTemps
            Group (59,302 187x110)
                Rectangle (0,0 150x30), "Warm"
                Lamp1 (155,0 30x30), variable: m_instance.stat.bWarm, style: Lamp-Lamp1-Blue
                Rectangle (2,40 150x30), "Partially Cold"
                Lamp1 (157,40 30x30), variable: m_instance.stat.bPartiallyCold, style: Lamp-Lamp1-Blue
                Rectangle (2,80 150x30), "Cold"
                Lamp1 (157,80 30x30), variable: m_instance.stat.bCold, style: Lamp-Lamp1-Blue
    Label (10,10 150x30), "Home"
    Group (248,40 545x110)
        Label (23,0 498x50), "METIS Cryo Controller"
        Rectangle (0,70 545x40), "%s", text variable: m_instance.stat.sState
    GroupBox (596,1020 420x177), "Evacuation"
        Rectangle (10,20 400x141), colour toggle: m_instance.stat.bEvacuationActive
        Group (16,33 135x30), invisible if: m_instance.stat.bEvacuationActive
            Lamp1 (105,0 30x30), variable: NOT m_instance.ctrl.bSafe_Evac, style: Lamp-Lamp1-Yellow
            Rectangle (0,0 100x30), "Interlock"
        Group (88,76 105x74)
            Group (0,44 105x30)
                Lamp1 (75,0 30x30), tooltip "If ON, TMP pump is at its nominal speed, i.e. Ready.", variable: m_Instance.met_evac.evac_branch_a.tp.stat.bReady, style: Lamp-Lamp1-Blue
                Rectangle (0,0 75x30), "TMP A"
            Group (0,0 105x30)
                Lamp1 (75,0 30x30), variable: m_Instance.met_evac.evac_branch_a.rp.stat.bReady, style: Lamp-Lamp1-Blue
                Rectangle (0,0 75x30), "PVP A"
        Group (256,76 105x74)
            Group (0,44 105x30)
                Lamp1 (75,0 30x30), tooltip "If ON, TMP pump is at its nominal speed, i.e. Ready.", variable: m_Instance.met_evac.evac_branch_b.tp.stat.bReady, style: Lamp-Lamp1-Blue
                Rectangle (0,0 75x30), "TMP B"
            Group (0,0 105x30)
                Lamp1 (75,0 30x30), variable: m_Instance.met_evac.evac_branch_b.rp.stat.bReady, style: Lamp-Lamp1-Blue
                Rectangle (0,0 75x30), "PVP B"
        Group (107,32 207x30)
            Rectangle (0,0 172x30), "Evacuation Active", invisible if: NOT m_instance.stat.bEvacuationActive
            Lamp1 (177,0 30x30), variable: m_instance.stat.bEvacuationActive, invisible if: NOT m_instance.stat.bEvacuationActive, style: Lamp-Lamp1-Green
    GroupBox (48,252 175x200)
        Group (13,13 142x156)
            Lamp1 (112,31 30x30), variable: m_instance.stat.bActive, style: Lamp-Lamp1-Green
            Rectangle (0,31 103x30), "Active"
            Rectangle (0,62 103x30), "Busy"
            Lamp1 (112,62 30x30), variable: m_instance.stat.bBusy, style: Lamp-Lamp1-Blue
            Rectangle (0,93 103x30), "Done"
            Lamp1 (112,93 30x30), variable: m_instance.stat.bDone, style: Lamp-Lamp1-Blue
            Lamp1 (112,126 30x30), variable: m_instance.stat.bError, style: Lamp-Lamp1-Red
            Rectangle (0,126 103x30), "Error"
            Lamp1 (112,0 30x30), variable: m_instance.stat.bInitialized, style: Lamp-Lamp1-Green
            Rectangle (0,0 103x30), "Initialized"
    GroupBox (732,180 290x357), "Cryostat Pressures"
        Group (40,32 210x315)
            Group (8,161 202x154)
                Group (15,0 185x30)
                    Rectangle (0,0 150x30), "Pressurized"
                    Lamp1 (155,0 30x30), variable: m_instance.stat.bPressurized, style: Lamp-Lamp1-Blue
                Group (17,41 185x30)
                    Rectangle (0,0 150x30), "Partial Vaccum"
                    Lamp1 (155,0 30x30), variable: m_instance.stat.bPartialVacuum, style: Lamp-Lamp1-Blue
                Group (0,82 202x30)
                    Rectangle (0,0 167x30), "Vacuum Achieved"
                    Lamp1 (172,0 30x30), variable: m_instance.stat.bInVacuum, style: Lamp-Lamp1-Blue
                Group (8,124 194x30)
                    Rectangle (0,0 159x30), "In Good Vacuum"
                    Lamp1 (164,0 30x30), variable: m_instance.stat.bInGoodVacuum, style: Lamp-Lamp1-Blue
            Group (0,0 210x141)
                Rectangle (85,0 125x35), "%.1e mbar", text variable: m_Instance.met_evac.VAGF.stat.lrPressure
                Rectangle (0,4 75x30), "VAGF"
                Rectangle (85,55 125x30), "%.1e mbar", text variable: m_Instance.met_evac.VAGG.stat.lrPressure
                Rectangle (0,57 75x30), "VAGG"
                Rectangle (85,109 125x30), "%.1e mbar", text variable: m_Instance.met_venting.HPG.stat.lrPressure
                Rectangle (0,111 75x30), "HPG"
    Frame (12,592 576x890)
        shows TEMPLATE_MAIN_FSM(m_instance := MAIN.met_cryo_ctrl)
    Frame (945,10 75x40)
        shows VISU_HMI_SUBSYSTEM_BUTTON(m_Hmi := PRG_HMI.fbBackButton)
        OnMouseClick: execute { PRG_HMI.eActiveTab := PRG_HMI.ePreviousTab; }
END_VISUALIZATION

// HMI/VISUs/ICS_Interlocks/VISU_HMI_ICS_INTERLOCKS
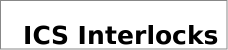
VISUALIZATION VISU_HMI_ICS_INTERLOCKS  // 228x50
    Label (20,20 208x30), "ICS Interlocks"
END_VISUALIZATION

// HMI/VISUs/Services/VISU_HMI_SERVICES
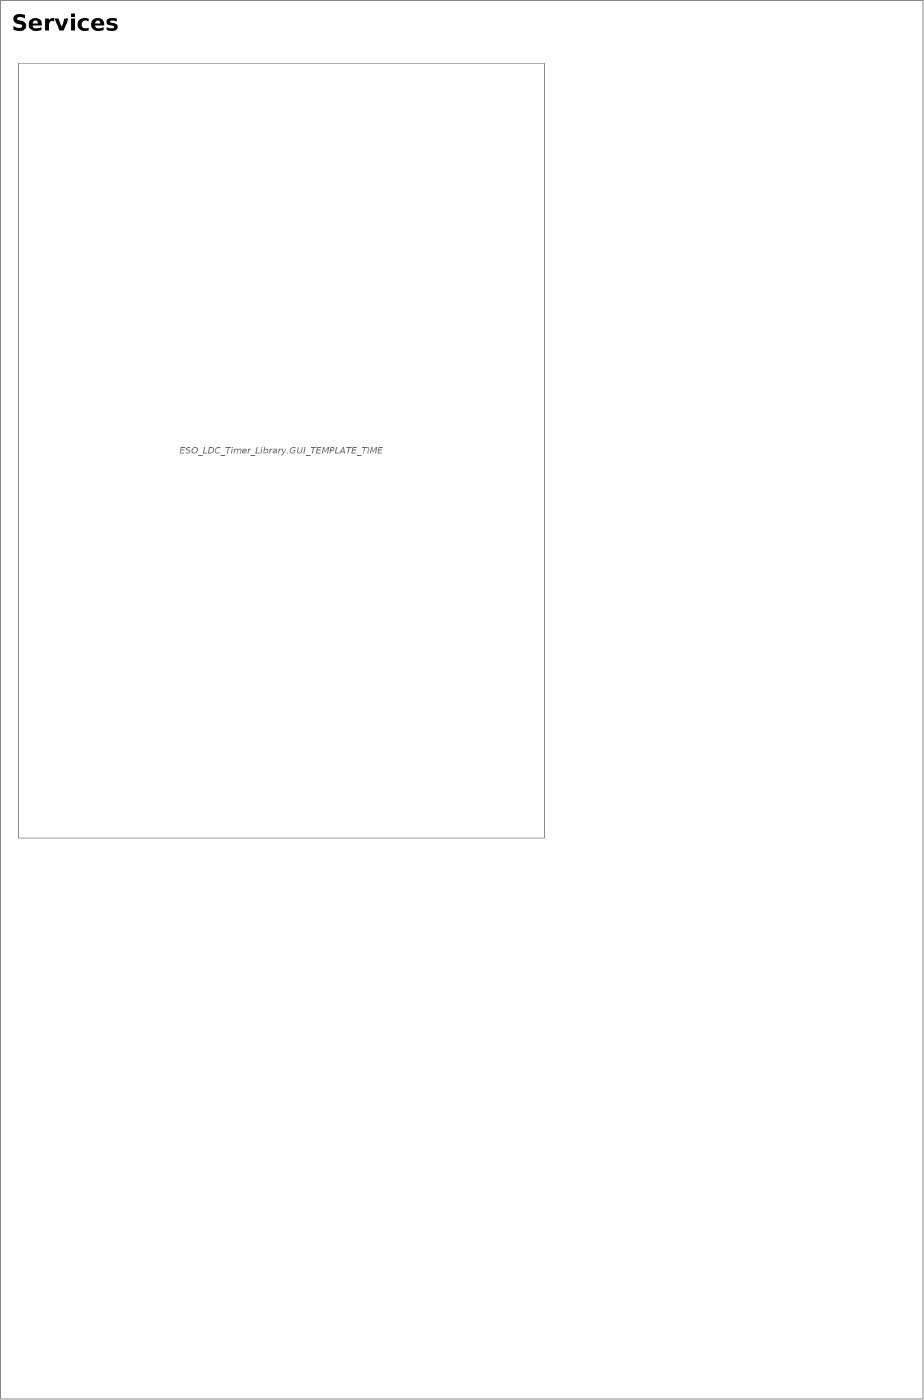
VISUALIZATION VISU_HMI_SERVICES  // 1030x1560
    Label (10,10 150x30), "Services"
    Frame (20,70 587x864)
        shows ESO_LDC_Timer_Library.GUI_TEMPLATE_TIME(m_Instance := MAIN.met_cryo_ctrl.met_cry_time)
END_VISUALIZATION

// HMI/VISUs/SIM_GUIs/GUI_Pressures_1
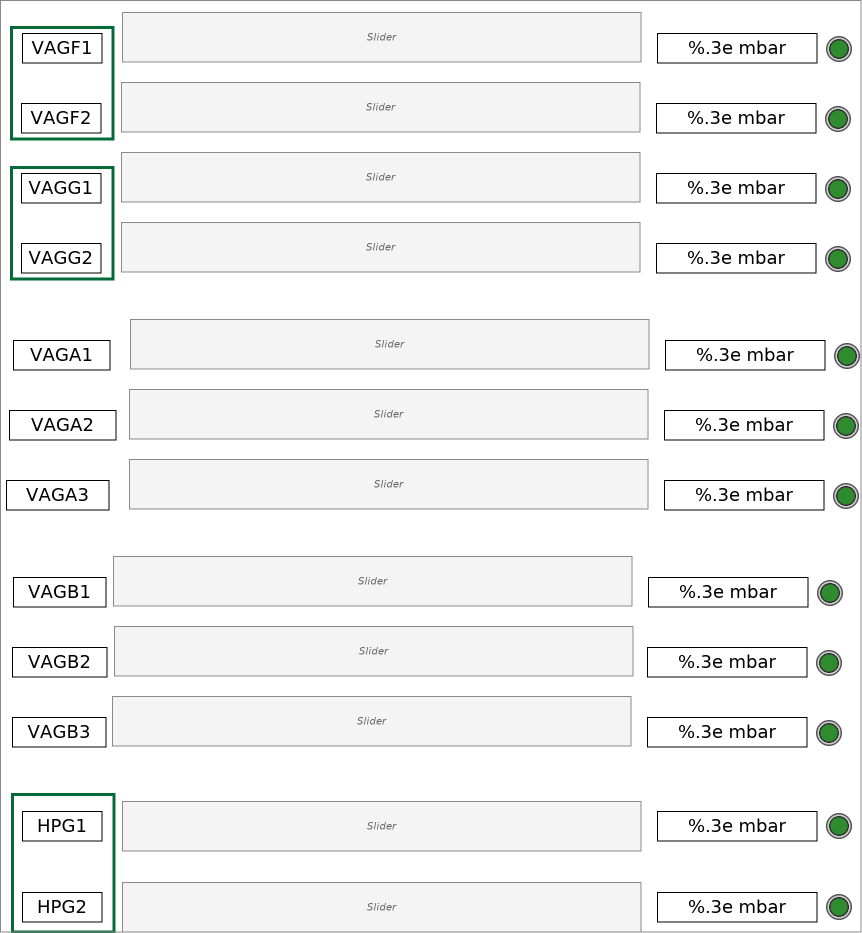
VISUALIZATION GUI_Pressures_1  // 862x933
VAR_IN_OUT
	m_instance:	FB_METIS_CRYO_EVAC;
	m_vent_instance: FB_METIS_CRYO_VENTING;
	
END_VAR
    Slider (130,319 519x50), variable: m_instance.q_nVAGA1, scale 0..35000
    Rectangle (13,340 97x30), "VAGA1"
    Rectangle (665,340 160x30), "%.3e mbar", text variable: m_instance.evac_branch_a.VAG1.stat.lrPressure
    Lamp1 (832,341 30x30), variable: m_instance.evac_branch_a.VAG1.stat.bValid, style: Lamp-Lamp1-Green
    Slider (129,389 519x50), variable: m_instance.q_nVAGA2, scale 0..35000
    Rectangle (9,410 107x30), "VAGA2"
    Rectangle (664,410 160x30), "%.3e mbar", text variable: m_instance.evac_branch_a.VAG2.stat.lrPressure
    Lamp1 (831,411 30x30), variable: m_instance.evac_branch_a.VAG2.stat.bValid, style: Lamp-Lamp1-Green
    Slider (129,459 519x50), variable: m_instance.q_nVAGA3, scale 0..35000
    Rectangle (6,480 103x30), "VAGA3"
    Rectangle (664,480 160x30), "%.3e mbar", text variable: m_instance.evac_branch_a.VAG3.stat.lrPressure
    Lamp1 (831,481 30x30), variable: m_instance.evac_branch_a.VAG3.stat.bValid, style: Lamp-Lamp1-Green
    Slider (122,12 519x50), variable: m_instance.q_nVAGF1, scale 0..35000
    Rectangle (22,33 80x30), "VAGF1"
    Rectangle (657,33 160x30), "%.3e mbar", text variable: m_instance.sensor_VAGF1.stat.lrPressure
    Lamp1 (824,34 30x30), variable: m_instance.sensor_VAGF1.stat.bValid, style: Lamp-Lamp1-Green
    Slider (121,82 519x50), variable: m_instance.q_nVAGF2, scale 0..35000
    Rectangle (21,103 80x30), "VAGF2"
    Rectangle (656,103 160x30), "%.3e mbar", text variable: m_instance.sensor_VAGF2.stat.lrPressure
    Lamp1 (823,104 30x30), variable: m_instance.sensor_VAGF2.stat.bValid, style: Lamp-Lamp1-Green
    Slider (121,152 519x50), variable: m_instance.q_nVAGG1, scale 0..35000
    Rectangle (21,173 80x30), "VAGG1"
    Rectangle (656,173 160x30), "%.3e mbar", text variable: m_instance.sensor_VAGG1.stat.lrPressure
    Lamp1 (823,174 30x30), variable: m_instance.sensor_VAGG1.stat.bValid, style: Lamp-Lamp1-Green
    Slider (121,222 519x50), variable: m_instance.q_nVAGG2, scale 0..35000
    Rectangle (21,243 80x30), "VAGG2"
    Rectangle (656,243 160x30), "%.3e mbar", text variable: m_instance.sensor_VAGG2.stat.lrPressure
    Lamp1 (823,244 30x30), variable: m_instance.sensor_VAGG2.stat.bValid, style: Lamp-Lamp1-Green
    Rectangle (10,26 104x114)
    Rectangle (10,166 104x114)
    Slider (113,556 519x50), variable: m_instance.q_nVAGB1, scale 0..35000
    Rectangle (13,577 93x30), "VAGB1"
    Rectangle (648,577 160x30), "%.3e mbar", text variable: m_instance.evac_branch_b.VAG1.stat.lrPressure
    Lamp1 (815,578 30x30), variable: m_instance.evac_branch_b.VAG1.stat.bValid, style: Lamp-Lamp1-Green
    Slider (114,626 519x50), variable: m_instance.q_nVAGB2, scale 0..35000
    Rectangle (12,647 95x30), "VAGB2"
    Rectangle (647,647 160x30), "%.3e mbar", text variable: m_instance.evac_branch_b.VAG2.stat.lrPressure
    Lamp1 (814,648 30x30), variable: m_instance.evac_branch_b.VAG2.stat.bValid, style: Lamp-Lamp1-Green
    Slider (112,696 519x50), variable: m_instance.q_nVAGB3, scale 0..35000
    Rectangle (12,717 94x30), "VAGB3"
    Rectangle (647,717 160x30), "%.3e mbar", text variable: m_instance.evac_branch_b.VAG3.stat.lrPressure
    Lamp1 (814,718 30x30), variable: m_instance.evac_branch_b.VAG3.stat.bValid, style: Lamp-Lamp1-Green
    Slider (122,801 519x50), variable: m_vent_instance.q_nSimHPG1, scale 0..35000
    Rectangle (22,811 80x30), "HPG1"
    Rectangle (657,811 160x30), "%.3e mbar", text variable: m_vent_instance.sensor_HPG1.stat.lrPressure
    Lamp1 (824,811 30x30), variable: m_vent_instance.sensor_HPG1.stat.bValid, style: Lamp-Lamp1-Green
    Slider (122,882 519x50), variable: m_vent_instance.q_nSimHPG2, scale 0..35000
    Rectangle (22,892 80x30), "HPG2"
    Rectangle (657,892 160x30), "%.3e mbar", text variable: m_vent_instance.sensor_HPG1.stat.lrPressure
    Rectangle (11,793 104x140)
    Lamp1 (824,892 30x30), variable: m_vent_instance.sensor_HPG2.stat.bValid, style: Lamp-Lamp1-Green
END_VISUALIZATION

// HMI/VISUs/SIM_GUIs/GUI_SIM_PRESSURES
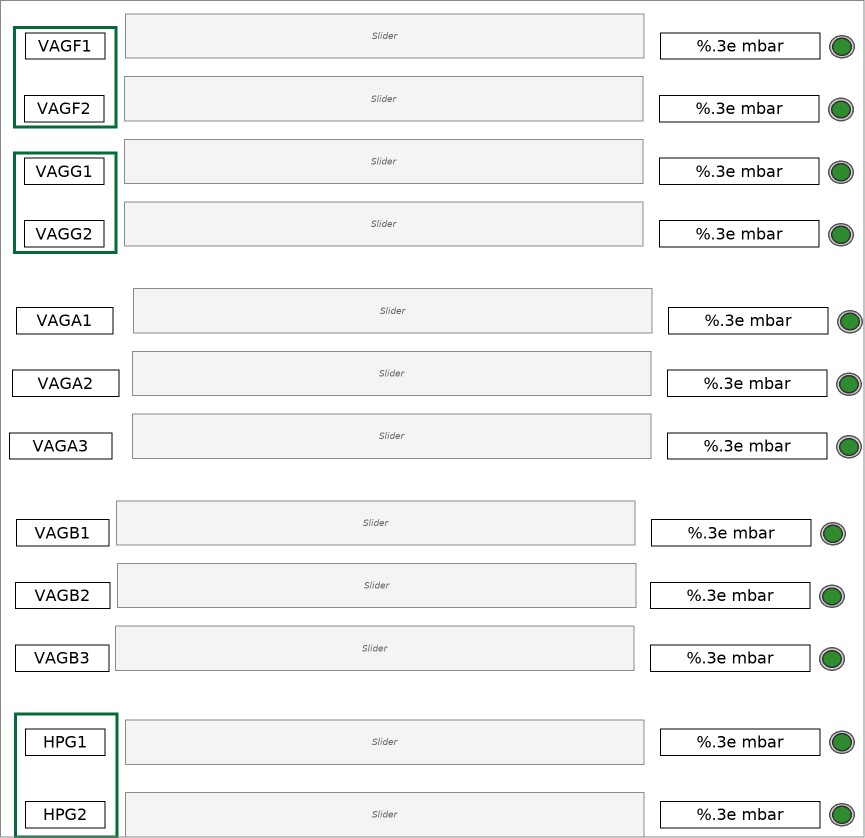
VISUALIZATION GUI_SIM_PRESSURES  // 865x838
    Frame (3,3 862x835)
        shows GUI_Pressures_1(m_instance := MAIN.met_cryo_ctrl.met_evac, m_vent_instance := MAIN.met_cryo_ctrl.met_venting)
END_VISUALIZATION

// HMI/VISUs/SIM_GUIs/GUI_SIM_SYSTEM_STATE
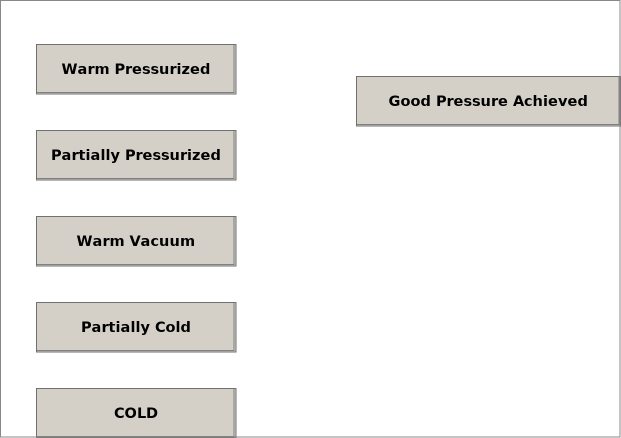
VISUALIZATION GUI_SIM_SYSTEM_STATE  // 621x438
    Button (36,44 200x50), "Warm Pressurized"
        OnMouseClick: execute {
            main.met_cryo_ctrl.stat.nState := E_METIS_CRYO_CTRL_STATE.WARM_PRESS;
            //Cry Temps
            main.met_cryo_ctrl.sim_lrHighestTemp 			:= 300;
            main.met_cryo_ctrl.sim_lrLowestTemp 			:= 300;
            main.met_cryo_ctrl.sim_lrCryostatTemp			:= 300;
            main.met_cryo_ctrl.sim_lrRadiationShielsTemp 	:= 300;
            // Ambient Temps
            main.met_cryo_ctrl.sim_lrDewPointTempC		:= 30;
            main.met_cryo_ctrl.sim_lrAmbiantTempC 		:= 30;
            main.met_cryo_ctrl.sim_lrWindowMountTempC 	:= 30;
            // Cry Pressures
            MAIN.met_cryo_ctrl.met_evac.q_nVAGF1 := 30000;
            MAIN.met_cryo_ctrl.met_evac.q_nVAGF2 := 30000;
            MAIN.met_cryo_ctrl.met_evac.q_nVAGG1 := 30000;
            MAIN.met_cryo_ctrl.met_evac.q_nVAGG2 := 30000;
            MAIN.met_cryo_ctrl.met_evac.q_nVAGA1 := 30000;
            MAIN.met_cryo_ctrl.met_evac.q_nVAGA2 := 30000;
            MAIN.met_cryo_ctrl.met_evac.q_nVAGA3 := 30000;
            MAIN.met_cryo_ctrl.met_evac.q_nVAGB1 := 30000;
            MAIN.met_cryo_ctrl.met_evac.q_nVAGB2 := 30000;
            MAIN.met_cryo_ctrl.met_evac.q_nVAGB3 := 30000;
            MAIN.met_cryo_ctrl.met_venting.q_nSimHPG1 := 30000;
            MAIN.met_cryo_ctrl.met_venting.q_nSimHPG2 := 30000;
        }
    Button (36,130 200x50), "Partially Pressurized"
        OnMouseClick: execute {
            main.met_cryo_ctrl.stat.nState := E_METIS_CRYO_CTRL_STATE.PARTIAL_VACUUM;
            //Cry Temps
            main.met_cryo_ctrl.sim_lrHighestTemp 			:= 300;
            main.met_cryo_ctrl.sim_lrLowestTemp 			:= 300;
            main.met_cryo_ctrl.sim_lrCryostatTemp			:= 300;
            main.met_cryo_ctrl.sim_lrRadiationShielsTemp 	:= 300;
            // Ambient Temps
            main.met_cryo_ctrl.sim_lrDewPointTempC		:= 30;
            main.met_cryo_ctrl.sim_lrAmbiantTempC 		:= 30;
            main.met_cryo_ctrl.sim_lrWindowMountTempC 	:= 30;
            // Cry Pressures
            MAIN.met_cryo_ctrl.met_evac.q_nVAGF1 := 27000;
            MAIN.met_cryo_ctrl.met_evac.q_nVAGF2 := 27000;
            MAIN.met_cryo_ctrl.met_evac.q_nVAGG1 := 27000;
            MAIN.met_cryo_ctrl.met_evac.q_nVAGG2 := 27000;
            MAIN.met_cryo_ctrl.met_evac.q_nVAGA1 := 27000;
            MAIN.met_cryo_ctrl.met_evac.q_nVAGA2 := 27000;
            MAIN.met_cryo_ctrl.met_evac.q_nVAGA3 := 27000;
            MAIN.met_cryo_ctrl.met_evac.q_nVAGB1 := 27000;
            MAIN.met_cryo_ctrl.met_evac.q_nVAGB2 := 27000;
            MAIN.met_cryo_ctrl.met_evac.q_nVAGB3 := 27000;
            MAIN.met_cryo_ctrl.met_venting.q_nSimHPG1 := 27000;
            MAIN.met_cryo_ctrl.met_venting.q_nSimHPG2 := 27000;
        }
    Button (36,216 200x50), "Warm Vacuum"
        OnMouseClick: execute {
            main.met_cryo_ctrl.stat.nState := E_METIS_CRYO_CTRL_STATE.WARM_VACUUM;
            //Cry Temps
            main.met_cryo_ctrl.sim_lrHighestTemp 			:= 300;
            main.met_cryo_ctrl.sim_lrLowestTemp 			:= 300;
            main.met_cryo_ctrl.sim_lrCryostatTemp			:= 300;
            main.met_cryo_ctrl.sim_lrRadiationShielsTemp 	:= 300;
            // Ambient Temps
            main.met_cryo_ctrl.sim_lrDewPointTempC		:= 30;
            main.met_cryo_ctrl.sim_lrAmbiantTempC 		:= 30;
            main.met_cryo_ctrl.sim_lrWindowMountTempC 	:= 30;
            // Cry Pressures
            MAIN.met_cryo_ctrl.met_evac.q_nVAGF1 := 16000;
            MAIN.met_cryo_ctrl.met_evac.q_nVAGF2 := 16000;
            MAIN.met_cryo_ctrl.met_evac.q_nVAGG1 := 16000;
            MAIN.met_cryo_ctrl.met_evac.q_nVAGG2 := 16000;
            MAIN.met_cryo_ctrl.met_evac.q_nVAGA1 := 16000;
            MAIN.met_cryo_ctrl.met_evac.q_nVAGA2 := 16000;
            MAIN.met_cryo_ctrl.met_evac.q_nVAGA3 := 16000;
            MAIN.met_cryo_ctrl.met_evac.q_nVAGB1 := 16000;
            MAIN.met_cryo_ctrl.met_evac.q_nVAGB2 := 16000;
            MAIN.met_cryo_ctrl.met_evac.q_nVAGB3 := 16000;
            MAIN.met_cryo_ctrl.met_venting.q_nSimHPG1 := 16000;
            MAIN.met_cryo_ctrl.met_venting.q_nSimHPG2 := 16000;
        }
    Button (356,76 265x50), "Good Pressure Achieved", tooltip "Only pressure values are modified"
        OnMouseClick: execute {
            // Cry Pressures
            MAIN.met_cryo_ctrl.met_evac.q_nVAGF1 := 11000;
            MAIN.met_cryo_ctrl.met_evac.q_nVAGF2 := 11000;
            MAIN.met_cryo_ctrl.met_evac.q_nVAGG1 := 11000;
            MAIN.met_cryo_ctrl.met_evac.q_nVAGG2 := 11000;
            MAIN.met_cryo_ctrl.met_evac.q_nVAGA1 := 11000;
            MAIN.met_cryo_ctrl.met_evac.q_nVAGA2 := 11000;
            MAIN.met_cryo_ctrl.met_evac.q_nVAGA3 := 11000;
            MAIN.met_cryo_ctrl.met_evac.q_nVAGB1 := 11000;
            MAIN.met_cryo_ctrl.met_evac.q_nVAGB2 := 11000;
            MAIN.met_cryo_ctrl.met_evac.q_nVAGB3 := 11000;
            MAIN.met_cryo_ctrl.met_venting.q_nSimHPG1 := 16000;
            MAIN.met_cryo_ctrl.met_venting.q_nSimHPG2 := 16000;
        }
    Button (36,302 200x50), "Partially Cold"
        OnMouseClick: execute {
            main.met_cryo_ctrl.stat.nState := E_METIS_CRYO_CTRL_STATE.PARTIALLY_COLD;
            //Cry Temps
            main.met_cryo_ctrl.sim_lrHighestTemp 			:= 250;
            main.met_cryo_ctrl.sim_lrLowestTemp 			:= 250;
            main.met_cryo_ctrl.sim_lrCryostatTemp			:= 250;
            main.met_cryo_ctrl.sim_lrRadiationShielsTemp 	:= 250;
            // Ambient Temps
            main.met_cryo_ctrl.sim_lrDewPointTempC		:= 30;
            main.met_cryo_ctrl.sim_lrAmbiantTempC 		:= 30;
            main.met_cryo_ctrl.sim_lrWindowMountTempC 	:= 30;
            // Cry Pressures
            MAIN.met_cryo_ctrl.met_evac.q_nVAGF1 := 16000;
            MAIN.met_cryo_ctrl.met_evac.q_nVAGF2 := 16000;
            MAIN.met_cryo_ctrl.met_evac.q_nVAGG1 := 16000;
            MAIN.met_cryo_ctrl.met_evac.q_nVAGG2 := 16000;
            MAIN.met_cryo_ctrl.met_evac.q_nVAGA1 := 16000;
            MAIN.met_cryo_ctrl.met_evac.q_nVAGA2 := 16000;
            MAIN.met_cryo_ctrl.met_evac.q_nVAGA3 := 16000;
            MAIN.met_cryo_ctrl.met_evac.q_nVAGB1 := 16000;
            MAIN.met_cryo_ctrl.met_evac.q_nVAGB2 := 16000;
            MAIN.met_cryo_ctrl.met_evac.q_nVAGB3 := 16000;
            MAIN.met_cryo_ctrl.met_venting.q_nSimHPG1 := 16000;
            MAIN.met_cryo_ctrl.met_venting.q_nSimHPG2 := 16000;
        }
    Button (36,388 200x50), "COLD"
        OnMouseClick: execute {
            main.met_cryo_ctrl.stat.nState := E_METIS_CRYO_CTRL_STATE.COLD;
            //Cry Temps
            main.met_cryo_ctrl.sim_lrHighestTemp 			:= 99;
            main.met_cryo_ctrl.sim_lrLowestTemp 			:= 99;
            main.met_cryo_ctrl.sim_lrCryostatTemp			:= 99;
            main.met_cryo_ctrl.sim_lrRadiationShielsTemp 	:= 99;
            // Ambient Temps
            main.met_cryo_ctrl.sim_lrDewPointTempC		:= 30;
            main.met_cryo_ctrl.sim_lrAmbiantTempC 		:= 30;
            main.met_cryo_ctrl.sim_lrWindowMountTempC 	:= 30;
            // Cry Pressures
            MAIN.met_cryo_ctrl.met_evac.q_nVAGF1 := 11000;
            MAIN.met_cryo_ctrl.met_evac.q_nVAGF2 := 11000;
            MAIN.met_cryo_ctrl.met_evac.q_nVAGG1 := 11000;
            MAIN.met_cryo_ctrl.met_evac.q_nVAGG2 := 11000;
            MAIN.met_cryo_ctrl.met_evac.q_nVAGA1 := 11000;
            MAIN.met_cryo_ctrl.met_evac.q_nVAGA2 := 11000;
            MAIN.met_cryo_ctrl.met_evac.q_nVAGA3 := 11000;
            MAIN.met_cryo_ctrl.met_evac.q_nVAGB1 := 11000;
            MAIN.met_cryo_ctrl.met_evac.q_nVAGB2 := 11000;
            MAIN.met_cryo_ctrl.met_evac.q_nVAGB3 := 11000;
            MAIN.met_cryo_ctrl.met_venting.q_nSimHPG1 := 11000;
            MAIN.met_cryo_ctrl.met_venting.q_nSimHPG2 := 11000;
        }
END_VISUALIZATION

// HMI/VISUs/SIM_GUIs/GUI_SIM_TEMPERATURES
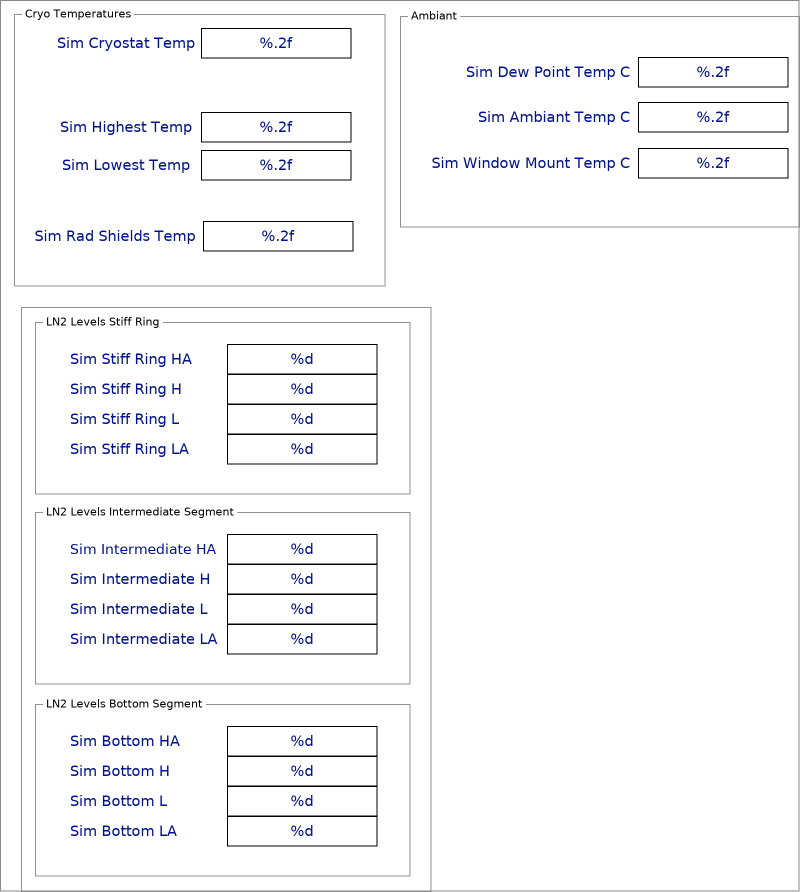
VISUALIZATION GUI_SIM_TEMPERATURES  // 800x892
    GroupBox (35,696 375x180), "LN2 Levels Bottom Segment"
        Rectangle (32,30 150x30), "Sim Bottom HA"
        Rectangle (192,30 150x30), "%d", tooltip "Simulated value [K] when simulation is active.", text variable: MAIN.met_cryo_ctrl.met_cool_down.nSim_LN2_LS_TempK[9]
            OnMouseClick: write the text variable via Default
        Rectangle (32,60 150x30), "Sim Bottom H"
        Rectangle (192,60 150x30), "%d", tooltip "Simulated value [K] when simulation is active.", text variable: MAIN.met_cryo_ctrl.met_cool_down.nSim_LN2_LS_TempK[10]
            OnMouseClick: write the text variable via Default
        Rectangle (32,90 150x30), "Sim Bottom L"
        Rectangle (192,90 150x30), "%d", tooltip "Simulated value [K] when simulation is active.", text variable: MAIN.met_cryo_ctrl.met_cool_down.nSim_LN2_LS_TempK[11]
            OnMouseClick: write the text variable via Default
        Rectangle (32,120 150x30), "Sim Bottom LA"
        Rectangle (192,120 150x30), "%d", tooltip "Simulated value [K] when simulation is active.", text variable: MAIN.met_cryo_ctrl.met_cool_down.nSim_LN2_LS_TempK[12]
            OnMouseClick: write the text variable via Default
    GroupBox (35,504 375x180), "LN2 Levels Intermediate Segment"
        Rectangle (32,30 150x30), "Sim Intermediate HA"
        Rectangle (192,30 150x30), "%d", tooltip "Simulated value [K] when simulation is active.", text variable: MAIN.met_cryo_ctrl.met_cool_down.nSim_LN2_LS_TempK[5]
            OnMouseClick: write the text variable via Default
        Rectangle (32,60 150x30), "Sim Intermediate H"
        Rectangle (192,60 150x30), "%d", tooltip "Simulated value [K] when simulation is active.", text variable: MAIN.met_cryo_ctrl.met_cool_down.nSim_LN2_LS_TempK[6]
            OnMouseClick: write the text variable via Default
        Rectangle (32,90 150x30), "Sim Intermediate L"
        Rectangle (192,90 150x30), "%d", tooltip "Simulated value [K] when simulation is active.", text variable: MAIN.met_cryo_ctrl.met_cool_down.nSim_LN2_LS_TempK[7]
            OnMouseClick: write the text variable via Default
        Rectangle (32,120 150x30), "Sim Intermediate LA"
        Rectangle (192,120 150x30), "%d", tooltip "Simulated value [K] when simulation is active.", text variable: MAIN.met_cryo_ctrl.met_cool_down.nSim_LN2_LS_TempK[8]
            OnMouseClick: write the text variable via Default
    Group (51,28 300x30)
        Rectangle (0,0 150x30), "Sim Cryostat Temp"
        Rectangle (150,0 150x30), "%.2f", tooltip "Simulated value [K] when simulation is active.", text variable: MAIN.met_cryo_ctrl.sim_lrCryostatTemp
            OnMouseClick: write the text variable via Default
    Group (51,112 300x30)
        Rectangle (0,0 150x30), "Sim Highest Temp"
        Rectangle (150,0 150x30), "%.2f", tooltip "Simulated value [K] when simulation is active.", text variable: MAIN.met_cryo_ctrl.sim_lrHighestTemp
            OnMouseClick: write the text variable via Default
    Group (51,150 300x30)
        Rectangle (0,0 150x30), "Sim Lowest Temp"
        Rectangle (150,0 150x30), "%.2f", tooltip "Simulated value [K] when simulation is active.", text variable: MAIN.met_cryo_ctrl.sim_lrLowestTemp
            OnMouseClick: write the text variable via Default
    Group (27,221 326x30)
        Rectangle (0,0 176x30), "Sim Rad Shields Temp"
        Rectangle (176,0 150x30), "%.2f", tooltip "Simulated value [K] when simulation is active.", text variable: MAIN.met_cryo_ctrl.sim_lrRadiationShielsTemp
            OnMouseClick: write the text variable via Default
    GroupBox (14,6 371x280), "Cryo Temperatures"
    GroupBox (400,8 400x219), "Ambiant"
        Group (13,49 375x30)
            Rectangle (0,0 220x30), "Sim Dew Point Temp C"
            Rectangle (225,0 150x30), "%.2f", tooltip "Simulated value [C] when simulation is active.", text variable: MAIN.met_cryo_ctrl.sim_lrDewPointTempC
                OnMouseClick: write the text variable via Default
        Group (13,94 375x30)
            Rectangle (0,0 220x30), "Sim Ambiant Temp C"
            Rectangle (225,0 150x30), "%.2f", tooltip "Simulated value [C] when simulation is active.", text variable: MAIN.met_cryo_ctrl.sim_lrAmbiantTempC
                OnMouseClick: write the text variable via Default
        Group (13,140 375x30)
            Rectangle (0,0 220x30), "Sim Window Mount Temp C"
            Rectangle (225,0 150x30), "%.2f", tooltip "Simulated value [C] when simulation is active.", text variable: MAIN.met_cryo_ctrl.sim_lrWindowMountTempC
                OnMouseClick: write the text variable via Default
    GroupBox (35,314 375x180), "LN2 Levels Stiff Ring"
    Rectangle (67,344 150x30), "Sim Stiff Ring HA"
    Rectangle (227,344 150x30), "%d", tooltip "Simulated value [K] when simulation is active.", text variable: MAIN.met_cryo_ctrl.met_cool_down.nSim_LN2_LS_TempK[1]
        OnMouseClick: write the text variable via Default
    Rectangle (67,374 150x30), "Sim Stiff Ring H"
    Rectangle (227,374 150x30), "%d", tooltip "Simulated value [K] when simulation is active.", text variable: MAIN.met_cryo_ctrl.met_cool_down.nSim_LN2_LS_TempK[2]
        OnMouseClick: write the text variable via Default
    Rectangle (67,404 150x30), "Sim Stiff Ring L"
    Rectangle (227,404 150x30), "%d", tooltip "Simulated value [K] when simulation is active.", text variable: MAIN.met_cryo_ctrl.met_cool_down.nSim_LN2_LS_TempK[3]
        OnMouseClick: write the text variable via Default
    Rectangle (67,434 150x30), "Sim Stiff Ring LA"
    Rectangle (227,434 150x30), "%d", tooltip "Simulated value [K] when simulation is active.", text variable: MAIN.met_cryo_ctrl.met_cool_down.nSim_LN2_LS_TempK[4]
        OnMouseClick: write the text variable via Default
    GroupBox (21,299 410x593)
END_VISUALIZATION

// HMI/VISUs/SIM_GUIs/VISU_SIM_PRESS_AND_TEMPS
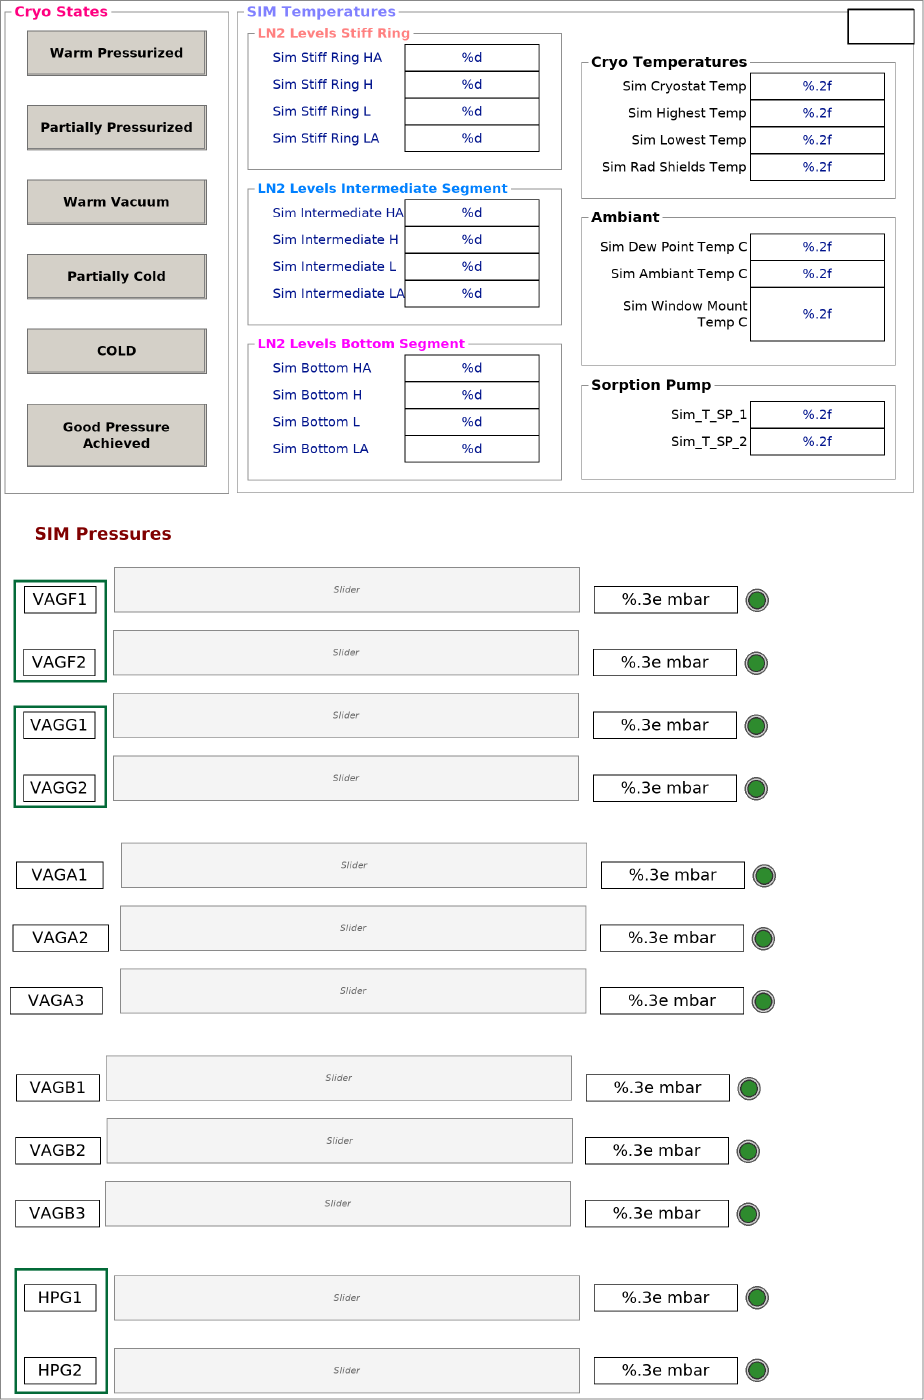
VISUALIZATION VISU_SIM_PRESS_AND_TEMPS  // 1030x1560
    GroupBox (264,5 754x544), "SIM Temperatures"
        Group (12,24 350x506)
            GroupBox (0,0 350x160), "LN2 Levels Stiff Ring"
                Group (25,20 300x120)
                    Group (0,90 300x30)
                        Rectangle (150,0 150x30), "%d", tooltip "Simulated value [K] when simulation is active.", text variable: MAIN.met_cryo_ctrl.met_cool_down.nSim_LN2_LS_TempK[4]
                            OnMouseClick: write the text variable via Default
                        Rectangle (0,0 150x30), "Sim Stiff Ring LA"
                    Group (0,60 300x30)
                        Rectangle (150,0 150x30), "%d", tooltip "Simulated value [K] when simulation is active.", text variable: MAIN.met_cryo_ctrl.met_cool_down.nSim_LN2_LS_TempK[3]
                            OnMouseClick: write the text variable via Default
                        Rectangle (0,0 150x30), "Sim Stiff Ring L"
                    Group (0,30 300x30)
                        Rectangle (150,0 150x30), "%d", tooltip "Simulated value [K] when simulation is active.", text variable: MAIN.met_cryo_ctrl.met_cool_down.nSim_LN2_LS_TempK[2]
                            OnMouseClick: write the text variable via Default
                        Rectangle (0,0 150x30), "Sim Stiff Ring H"
                    Group (0,0 300x30)
                        Rectangle (150,0 150x30), "%d", tooltip "Simulated value [K] when simulation is active.", text variable: MAIN.met_cryo_ctrl.met_cool_down.nSim_LN2_LS_TempK[1]
                            OnMouseClick: write the text variable via Default
                        Rectangle (0,0 150x30), "Sim Stiff Ring HA"
            GroupBox (0,173 350x160), "LN2 Levels Intermediate Segment"
                Group (25,20 300x120)
                    Group (0,0 300x30)
                        Rectangle (0,0 150x30), "Sim Intermediate HA"
                        Rectangle (150,0 150x30), "%d", tooltip "Simulated value [K] when simulation is active.", text variable: MAIN.met_cryo_ctrl.met_cool_down.nSim_LN2_LS_TempK[5]
                            OnMouseClick: write the text variable via Default
                    Group (0,30 300x30)
                        Rectangle (0,0 150x30), "Sim Intermediate H"
                        Rectangle (150,0 150x30), "%d", tooltip "Simulated value [K] when simulation is active.", text variable: MAIN.met_cryo_ctrl.met_cool_down.nSim_LN2_LS_TempK[6]
                            OnMouseClick: write the text variable via Default
                    Group (0,60 300x30)
                        Rectangle (0,0 150x30), "Sim Intermediate L"
                        Rectangle (150,0 150x30), "%d", tooltip "Simulated value [K] when simulation is active.", text variable: MAIN.met_cryo_ctrl.met_cool_down.nSim_LN2_LS_TempK[7]
                            OnMouseClick: write the text variable via Default
                    Group (0,90 300x30)
                        Rectangle (0,0 150x30), "Sim Intermediate LA"
                        Rectangle (150,0 150x30), "%d", tooltip "Simulated value [K] when simulation is active.", text variable: MAIN.met_cryo_ctrl.met_cool_down.nSim_LN2_LS_TempK[8]
                            OnMouseClick: write the text variable via Default
            GroupBox (0,346 350x160), "LN2 Levels Bottom Segment"
                Group (25,20 300x120)
                    Group (0,0 300x30)
                        Rectangle (0,0 150x30), "Sim Bottom HA"
                        Rectangle (150,0 150x30), "%d", tooltip "Simulated value [K] when simulation is active.", text variable: MAIN.met_cryo_ctrl.met_cool_down.nSim_LN2_LS_TempK[9]
                            OnMouseClick: write the text variable via Default
                    Group (0,30 300x30)
                        Rectangle (0,0 150x30), "Sim Bottom H"
                        Rectangle (150,0 150x30), "%d", tooltip "Simulated value [K] when simulation is active.", text variable: MAIN.met_cryo_ctrl.met_cool_down.nSim_LN2_LS_TempK[10]
                            OnMouseClick: write the text variable via Default
                    Group (0,60 300x30)
                        Rectangle (0,0 150x30), "Sim Bottom L"
                        Rectangle (150,0 150x30), "%d", tooltip "Simulated value [K] when simulation is active.", text variable: MAIN.met_cryo_ctrl.met_cool_down.nSim_LN2_LS_TempK[11]
                            OnMouseClick: write the text variable via Default
                    Group (0,90 300x30)
                        Rectangle (0,0 150x30), "Sim Bottom LA"
                        Rectangle (150,0 150x30), "%d", tooltip "Simulated value [K] when simulation is active.", text variable: MAIN.met_cryo_ctrl.met_cool_down.nSim_LN2_LS_TempK[12]
                            OnMouseClick: write the text variable via Default
        GroupBox (384,229 350x173), "Ambiant"
            Group (13,26 325x120)
                Group (0,0 325x30)
                    Rectangle (0,0 175x30), "Sim Dew Point Temp C"
                    Rectangle (175,0 150x30), "%.2f", tooltip "Simulated value [C] when simulation is active.", text variable: MAIN.met_cryo_ctrl.sim_lrDewPointTempC
                        OnMouseClick: write the text variable via Default
                Group (0,30 325x30)
                    Rectangle (0,0 175x30), "Sim Ambiant Temp C"
                    Rectangle (175,0 150x30), "%.2f", tooltip "Simulated value [C] when simulation is active.", text variable: MAIN.met_cryo_ctrl.sim_lrAmbiantTempC
                        OnMouseClick: write the text variable via Default
                Group (0,60 325x60)
                    Rectangle (0,0 175x60), "Sim Window Mount Temp C"
                    Rectangle (175,0 150x60), "%.2f", tooltip "Simulated value [C] when simulation is active.", text variable: MAIN.met_cryo_ctrl.sim_lrWindowMountTempC
                        OnMouseClick: write the text variable via Default
        GroupBox (384,56 350x160), "Cryo Temperatures"
            Group (12,20 326x120)
                Group (0,0 326x30)
                    Rectangle (0,0 175x30), "Sim Cryostat Temp"
                    Rectangle (176,0 150x30), "%.2f", tooltip "Simulated value [K] when simulation is active.", text variable: MAIN.met_cryo_ctrl.sim_lrCryostatTemp
                        OnMouseClick: write the text variable via Default
                Group (0,30 326x30)
                    Rectangle (0,0 175x30), "Sim Highest Temp"
                    Rectangle (176,0 150x30), "%.2f", tooltip "Simulated value [K] when simulation is active.", text variable: MAIN.met_cryo_ctrl.sim_lrHighestTemp
                        OnMouseClick: write the text variable via Default
                Group (0,60 326x30)
                    Rectangle (0,0 175x30), "Sim Lowest Temp"
                    Rectangle (176,0 150x30), "%.2f", tooltip "Simulated value [K] when simulation is active.", text variable: MAIN.met_cryo_ctrl.sim_lrLowestTemp
                        OnMouseClick: write the text variable via Default
                Group (0,90 326x30)
                    Rectangle (0,0 175x30), "Sim Rad Shields Temp"
                    Rectangle (176,0 150x30), "%.2f", tooltip "Simulated value [K] when simulation is active.", text variable: MAIN.met_cryo_ctrl.sim_lrRadiationShielsTemp
                        OnMouseClick: write the text variable via Default
        GroupBox (384,416 350x113), "Sorption Pump"
            Rectangle (13,26 175x30), "Sim_T_SP_1"
            Rectangle (188,26 150x30), "%.2f", tooltip "Simulated SP 1 temp value [K]", text variable: MAIN.met_cryo_ctrl.sim_regeneration.sim_t_sp_1
                OnMouseClick: write the text variable via Default
            Rectangle (13,56 175x30), "Sim_T_SP_2"
            Rectangle (188,56 150x30), "%.2f", tooltip "Simulated SP 2 temp value [K]", text variable: MAIN.met_cryo_ctrl.sim_regeneration.sim_t_sp_2
                OnMouseClick: write the text variable via Default
    GroupBox (5,5 250x545), "Cryo States", tooltip "Cryo states"
        Group (25,29 200x486)
            Button (0,0 200x50), "Warm Pressurized"
                OnMouseClick: execute {
                    main.met_cryo_ctrl.stat.nState := E_METIS_CRYO_CTRL_STATE.WARM_PRESS;
                    //Cry Temps
                    main.met_cryo_ctrl.sim_lrHighestTemp 			:= 300;
                    main.met_cryo_ctrl.sim_lrLowestTemp 			:= 300;
                    main.met_cryo_ctrl.sim_lrCryostatTemp			:= 300;
                    main.met_cryo_ctrl.sim_lrRadiationShielsTemp 	:= 300;
                    // Ambient Temps
                    main.met_cryo_ctrl.sim_lrDewPointTempC		:= 30;
                    main.met_cryo_ctrl.sim_lrAmbiantTempC 		:= 30;
                    main.met_cryo_ctrl.sim_lrWindowMountTempC 	:= 30;
                    // Cry Pressures
                    MAIN.met_cryo_ctrl.met_evac.q_nVAGF1 := 30000;
                    MAIN.met_cryo_ctrl.met_evac.q_nVAGF2 := 30000;
                    MAIN.met_cryo_ctrl.met_evac.q_nVAGG1 := 30000;
                    MAIN.met_cryo_ctrl.met_evac.q_nVAGG2 := 30000;
                    MAIN.met_cryo_ctrl.met_evac.q_nVAGA1 := 30000;
                    MAIN.met_cryo_ctrl.met_evac.q_nVAGA2 := 30000;
                    MAIN.met_cryo_ctrl.met_evac.q_nVAGA3 := 30000;
                    MAIN.met_cryo_ctrl.met_evac.q_nVAGB1 := 30000;
                    MAIN.met_cryo_ctrl.met_evac.q_nVAGB2 := 30000;
                    MAIN.met_cryo_ctrl.met_evac.q_nVAGB3 := 30000;
                    MAIN.met_cryo_ctrl.met_venting.q_nSimHPG1 := 30000;
                    MAIN.met_cryo_ctrl.met_venting.q_nSimHPG2 := 30000;
                }
            Button (0,83 200x50), "Partially Pressurized"
                OnMouseClick: execute {
                    main.met_cryo_ctrl.stat.nState := E_METIS_CRYO_CTRL_STATE.PARTIAL_VACUUM;
                    //Cry Temps
                    main.met_cryo_ctrl.sim_lrHighestTemp 			:= 300;
                    main.met_cryo_ctrl.sim_lrLowestTemp 			:= 300;
                    main.met_cryo_ctrl.sim_lrCryostatTemp			:= 300;
                    main.met_cryo_ctrl.sim_lrRadiationShielsTemp 	:= 300;
                    // Ambient Temps
                    main.met_cryo_ctrl.sim_lrDewPointTempC		:= 30;
                    main.met_cryo_ctrl.sim_lrAmbiantTempC 		:= 30;
                    main.met_cryo_ctrl.sim_lrWindowMountTempC 	:= 30;
                    // Cry Pressures
                    MAIN.met_cryo_ctrl.met_evac.q_nVAGF1 := 27000;
                    MAIN.met_cryo_ctrl.met_evac.q_nVAGF2 := 27000;
                    MAIN.met_cryo_ctrl.met_evac.q_nVAGG1 := 27000;
                    MAIN.met_cryo_ctrl.met_evac.q_nVAGG2 := 27000;
                    MAIN.met_cryo_ctrl.met_evac.q_nVAGA1 := 27000;
                    MAIN.met_cryo_ctrl.met_evac.q_nVAGA2 := 27000;
                    MAIN.met_cryo_ctrl.met_evac.q_nVAGA3 := 27000;
                    MAIN.met_cryo_ctrl.met_evac.q_nVAGB1 := 27000;
                    MAIN.met_cryo_ctrl.met_evac.q_nVAGB2 := 27000;
                    MAIN.met_cryo_ctrl.met_evac.q_nVAGB3 := 27000;
                    MAIN.met_cryo_ctrl.met_venting.q_nSimHPG1 := 27000;
                    MAIN.met_cryo_ctrl.met_venting.q_nSimHPG2 := 27000;
                }
            Button (0,166 200x50), "Warm Vacuum"
                OnMouseClick: execute {
                    main.met_cryo_ctrl.stat.nState := E_METIS_CRYO_CTRL_STATE.WARM_VACUUM;
                    //Cry Temps
                    main.met_cryo_ctrl.sim_lrHighestTemp 			:= 300;
                    main.met_cryo_ctrl.sim_lrLowestTemp 			:= 300;
                    main.met_cryo_ctrl.sim_lrCryostatTemp			:= 300;
                    main.met_cryo_ctrl.sim_lrRadiationShielsTemp 	:= 300;
                    // Ambient Temps
                    main.met_cryo_ctrl.sim_lrDewPointTempC		:= 30;
                    main.met_cryo_ctrl.sim_lrAmbiantTempC 		:= 30;
                    main.met_cryo_ctrl.sim_lrWindowMountTempC 	:= 30;
                    // Cry Pressures
                    MAIN.met_cryo_ctrl.met_evac.q_nVAGF1 := 16000;
                    MAIN.met_cryo_ctrl.met_evac.q_nVAGF2 := 16000;
                    MAIN.met_cryo_ctrl.met_evac.q_nVAGG1 := 16000;
                    MAIN.met_cryo_ctrl.met_evac.q_nVAGG2 := 16000;
                    MAIN.met_cryo_ctrl.met_evac.q_nVAGA1 := 16000;
                    MAIN.met_cryo_ctrl.met_evac.q_nVAGA2 := 16000;
                    MAIN.met_cryo_ctrl.met_evac.q_nVAGA3 := 16000;
                    MAIN.met_cryo_ctrl.met_evac.q_nVAGB1 := 16000;
                    MAIN.met_cryo_ctrl.met_evac.q_nVAGB2 := 16000;
                    MAIN.met_cryo_ctrl.met_evac.q_nVAGB3 := 16000;
                    MAIN.met_cryo_ctrl.met_venting.q_nSimHPG1 := 16000;
                    MAIN.met_cryo_ctrl.met_venting.q_nSimHPG2 := 16000;
                }
            Button (0,416 200x70), "Good Pressure Achieved", tooltip "Only pressure values are modified"
                OnMouseClick: execute {
                    // Cry Pressures
                    MAIN.met_cryo_ctrl.met_evac.q_nVAGF1 := 11000;
                    MAIN.met_cryo_ctrl.met_evac.q_nVAGF2 := 11000;
                    MAIN.met_cryo_ctrl.met_evac.q_nVAGG1 := 11000;
                    MAIN.met_cryo_ctrl.met_evac.q_nVAGG2 := 11000;
                    MAIN.met_cryo_ctrl.met_evac.q_nVAGA1 := 11000;
                    MAIN.met_cryo_ctrl.met_evac.q_nVAGA2 := 11000;
                    MAIN.met_cryo_ctrl.met_evac.q_nVAGA3 := 11000;
                    MAIN.met_cryo_ctrl.met_evac.q_nVAGB1 := 11000;
                    MAIN.met_cryo_ctrl.met_evac.q_nVAGB2 := 11000;
                    MAIN.met_cryo_ctrl.met_evac.q_nVAGB3 := 11000;
                    MAIN.met_cryo_ctrl.met_venting.q_nSimHPG1 := 16000;
                    MAIN.met_cryo_ctrl.met_venting.q_nSimHPG2 := 16000;
                }
            Button (0,249 200x50), "Partially Cold"
                OnMouseClick: execute {
                    main.met_cryo_ctrl.stat.nState := E_METIS_CRYO_CTRL_STATE.PARTIALLY_COLD;
                    //Cry Temps
                    main.met_cryo_ctrl.sim_lrHighestTemp 			:= 250;
                    main.met_cryo_ctrl.sim_lrLowestTemp 			:= 250;
                    main.met_cryo_ctrl.sim_lrCryostatTemp			:= 250;
                    main.met_cryo_ctrl.sim_lrRadiationShielsTemp 	:= 250;
                    // Ambient Temps
                    main.met_cryo_ctrl.sim_lrDewPointTempC		:= 30;
                    main.met_cryo_ctrl.sim_lrAmbiantTempC 		:= 30;
                    main.met_cryo_ctrl.sim_lrWindowMountTempC 	:= 30;
                    // Cry Pressures
                    MAIN.met_cryo_ctrl.met_evac.q_nVAGF1 := 16000;
                    MAIN.met_cryo_ctrl.met_evac.q_nVAGF2 := 16000;
                    MAIN.met_cryo_ctrl.met_evac.q_nVAGG1 := 16000;
                    MAIN.met_cryo_ctrl.met_evac.q_nVAGG2 := 16000;
                    MAIN.met_cryo_ctrl.met_evac.q_nVAGA1 := 16000;
                    MAIN.met_cryo_ctrl.met_evac.q_nVAGA2 := 16000;
                    MAIN.met_cryo_ctrl.met_evac.q_nVAGA3 := 16000;
                    MAIN.met_cryo_ctrl.met_evac.q_nVAGB1 := 16000;
                    MAIN.met_cryo_ctrl.met_evac.q_nVAGB2 := 16000;
                    MAIN.met_cryo_ctrl.met_evac.q_nVAGB3 := 16000;
                    MAIN.met_cryo_ctrl.met_venting.q_nSimHPG1 := 16000;
                    MAIN.met_cryo_ctrl.met_venting.q_nSimHPG2 := 16000;
                }
            Button (0,332 200x50), "COLD"
                OnMouseClick: execute {
                    main.met_cryo_ctrl.stat.nState := E_METIS_CRYO_CTRL_STATE.COLD;
                    //Cry Temps
                    main.met_cryo_ctrl.sim_lrHighestTemp 			:= 99;
                    main.met_cryo_ctrl.sim_lrLowestTemp 			:= 99;
                    main.met_cryo_ctrl.sim_lrCryostatTemp			:= 99;
                    main.met_cryo_ctrl.sim_lrRadiationShielsTemp 	:= 99;
                    // Ambient Temps
                    main.met_cryo_ctrl.sim_lrDewPointTempC		:= 30;
                    main.met_cryo_ctrl.sim_lrAmbiantTempC 		:= 30;
                    main.met_cryo_ctrl.sim_lrWindowMountTempC 	:= 30;
                    // Cry Pressures
                    MAIN.met_cryo_ctrl.met_evac.q_nVAGF1 := 11000;
                    MAIN.met_cryo_ctrl.met_evac.q_nVAGF2 := 11000;
                    MAIN.met_cryo_ctrl.met_evac.q_nVAGG1 := 11000;
                    MAIN.met_cryo_ctrl.met_evac.q_nVAGG2 := 11000;
                    MAIN.met_cryo_ctrl.met_evac.q_nVAGA1 := 11000;
                    MAIN.met_cryo_ctrl.met_evac.q_nVAGA2 := 11000;
                    MAIN.met_cryo_ctrl.met_evac.q_nVAGA3 := 11000;
                    MAIN.met_cryo_ctrl.met_evac.q_nVAGB1 := 11000;
                    MAIN.met_cryo_ctrl.met_evac.q_nVAGB2 := 11000;
                    MAIN.met_cryo_ctrl.met_evac.q_nVAGB3 := 11000;
                    MAIN.met_cryo_ctrl.met_venting.q_nSimHPG1 := 11000;
                    MAIN.met_cryo_ctrl.met_venting.q_nSimHPG2 := 11000;
                }
    Frame (5,620 862x935)
        shows GUI_Pressures_1(m_instance := MAIN.met_cryo_ctrl.met_evac, m_vent_instance := MAIN.met_cryo_ctrl.met_venting)
    Rectangle (12,580 206x30), "SIM Pressures"
    Frame (945,10 75x40)
        shows VISU_HMI_SUBSYSTEM_BUTTON(m_Hmi := PRG_HMI.fbBackButton)
        OnMouseClick: execute { PRG_HMI.eActiveTab := PRG_HMI.ePreviousTab; }
END_VISUALIZATION

// HMI/VISUs/Subsystems/CFO/VISU_HMI_CFO
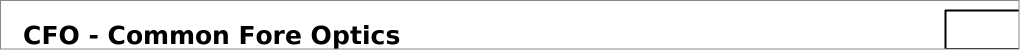
VISUALIZATION VISU_HMI_CFO  // 1020x50
    Label (20,20 671x30), "CFO - Common Fore Optics"
    Frame (945,10 75x40)
        shows VISU_HMI_SUBSYSTEM_BUTTON(m_Hmi := PRG_HMI.fbBackButton)
        OnMouseClick: execute { PRG_HMI.eActiveTab := PRG_HMI.ePreviousTab; }
END_VISUALIZATION

// HMI/VISUs/Subsystems/CRY/Components/VISU_HMI_CRY_HEATERS
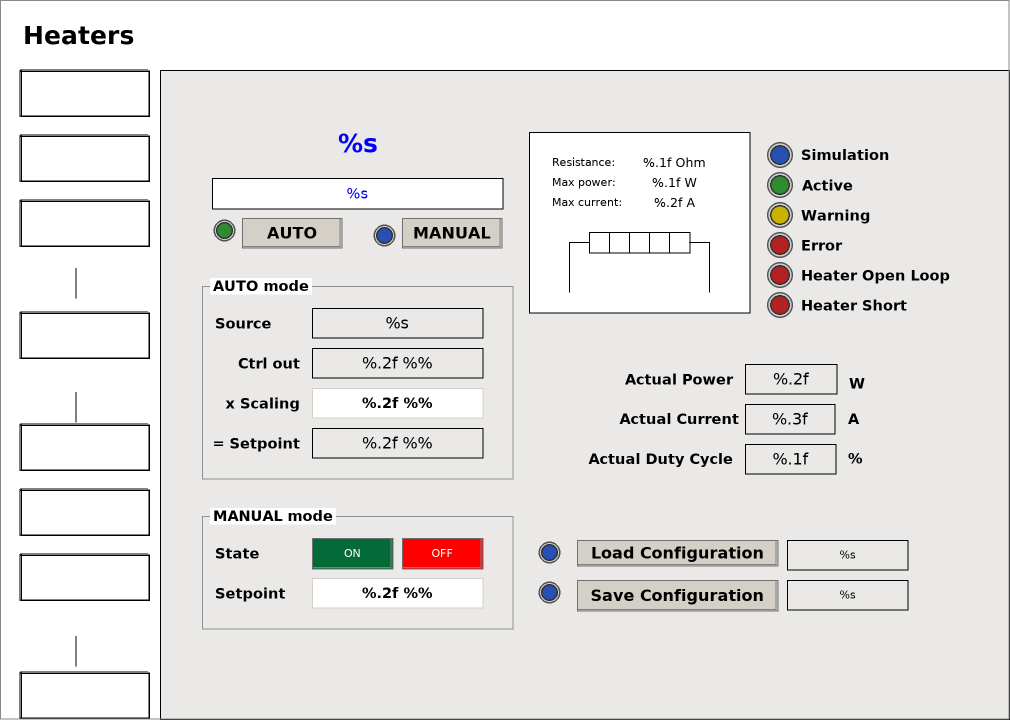
VISUALIZATION VISU_HMI_CRY_HEATERS  // 1010x720
VAR_IN_OUT
	m_Instance : FB_METIS_HEATERS;
    m_Hmi : FB_HMI_CRY_HEATERS;
END_VAR
    Rectangle (160,70 850x650)
    Frame (185,120 800x550), frame switch variable: m_Hmi.eActiveTab
        shows TEMPLATE_METIS_HEATER(m_instance := m_Instance.h_cry_sha)
        shows TEMPLATE_METIS_HEATER(m_instance := m_Instance.h_cry_shb)
        shows TEMPLATE_METIS_HEATER(m_instance := m_Instance.h_cry_shc)
        shows TEMPLATE_METIS_HEATER(m_instance := m_Instance.h_cry_sp)
        shows TEMPLATE_METIS_HEATER(m_instance := m_Instance.h_cry_pta)
        shows TEMPLATE_METIS_HEATER(m_instance := m_Instance.h_cry_ptb)
        shows TEMPLATE_METIS_HEATER(m_instance := m_Instance.h_cry_ptc)
        shows TEMPLATE_METIS_HEATER(m_instance := m_Instance.h_cry_wi)
        p8630679: tcontrol.tc_img_wuh_1
        p371692913: tcontrol.vote_img_wuh_1
        p2286783886: temperatures
    Frame (20,70 131x48)
        shows VISU_HMI_SUBSYSTEM_BUTTON(m_Hmi := m_Hmi.h_cry_sha_button)
        OnMouseClick: execute { m_Hmi.eActiveTab := E_HMI_CRY_HEATER_TABS.H_CRY_SHA; }
    Frame (20,135 131x48)
        shows VISU_HMI_SUBSYSTEM_BUTTON(m_Hmi := m_Hmi.h_cry_shb_button)
        OnMouseClick: execute { m_Hmi.eActiveTab := E_HMI_CRY_HEATER_TABS.H_CRY_SHB; }
    Frame (20,200 131x48)
        shows VISU_HMI_SUBSYSTEM_BUTTON(m_Hmi := m_Hmi.h_cry_shc_button)
        OnMouseClick: execute { m_Hmi.eActiveTab := E_HMI_CRY_HEATER_TABS.H_CRY_SHC; }
    Frame (20,312 131x48)
        shows VISU_HMI_SUBSYSTEM_BUTTON(m_Hmi := m_Hmi.h_cry_sp_button)
        OnMouseClick: execute { m_Hmi.eActiveTab := E_HMI_CRY_HEATER_TABS.H_CRY_SP; }
    Line (76,298) (76,268)
    Line (76,422) (76,392)
    Frame (20,424 131x48)
        shows VISU_HMI_SUBSYSTEM_BUTTON(m_Hmi := m_Hmi.h_cry_pta_button)
        OnMouseClick: execute { m_Hmi.eActiveTab := E_HMI_CRY_HEATER_TABS.H_CRY_PTA; }
    Frame (20,489 131x48)
        shows VISU_HMI_SUBSYSTEM_BUTTON(m_Hmi := m_Hmi.h_cry_ptb_button)
        OnMouseClick: execute { m_Hmi.eActiveTab := E_HMI_CRY_HEATER_TABS.H_CRY_PTB; }
    Frame (20,554 131x48)
        shows VISU_HMI_SUBSYSTEM_BUTTON(m_Hmi := m_Hmi.h_cry_ptc_button)
        OnMouseClick: execute { m_Hmi.eActiveTab := E_HMI_CRY_HEATER_TABS.H_CRY_PTC; }
    Frame (20,672 131x48)
        shows VISU_HMI_SUBSYSTEM_BUTTON(m_Hmi := m_Hmi.h_cry_wi_button)
        OnMouseClick: execute { m_Hmi.eActiveTab := E_HMI_CRY_HEATER_TABS.H_CRY_WI; }
    Line (76,666) (76,636)
    Label (20,20 411x30), "Heaters"
END_VISUALIZATION

// HMI/VISUs/Subsystems/CRY/Components/VISU_HMI_CRY_LN2_LEVEL_CONTROL
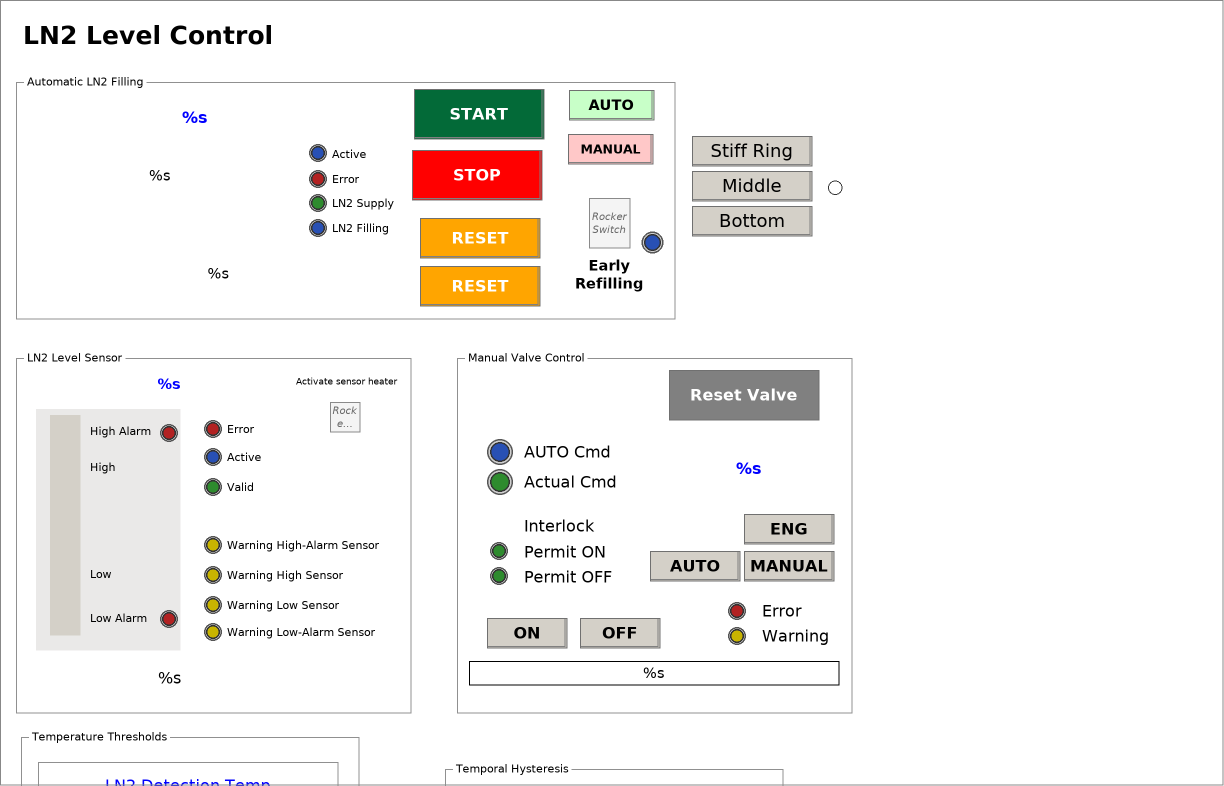
VISUALIZATION VISU_HMI_CRY_LN2_LEVEL_CONTROL  // 1224x786
    Label (20,20 299x30), "LN2 Level Control"
    Frame (0,70 1224x716)
        shows TEMPLATE_LN2_LEVEL_SENSOR_AND_CTRL(m_level_control_instance := MAIN.met_cryo_ctrl.met_cool_down.lc_ln2_level_ctrl[MAIN.met_cryo_ctrl.met_cool_down.gui_index_ln2_ctrl], m_instance := MAIN.met_cryo_ctrl.met_cool_down.lc_ln2_level_ctrl[MAIN.met_cryo_ctrl.met_cool_down.gui_index_ln2_ctrl].LN2_Level, m_cmd := MAIN.met_cryo_ctrl.met_cool_down.lc_ln2_level_ctrl[MAIN.met_cryo_ctrl.met_cool_down.gui_index_ln2_ctrl].cor_ln2_level_ctrl, m_bEnable := MAIN.met_cryo_ctrl.met_cool_down.lc_ln2_level_ctrl[MAIN.met_cryo_ctrl.met_cool_down.gui_index_ln2_ctrl].bEnable)
    Group (692,136 167x103)
        Button (0,0 120x30), "Stiff Ring", tooltip "Shield A"
            OnMouseClick: execute { MAIN.met_cryo_ctrl.met_cool_down.gui_index_ln2_ctrl := 1; }
        Button (0,35 120x30), "Middle", tooltip "Shield B"
            OnMouseClick: execute { MAIN.met_cryo_ctrl.met_cool_down.gui_index_ln2_ctrl := 2; }
        Button (0,70 120x30), "Bottom", tooltip "Shield C"
            OnMouseClick: execute { MAIN.met_cryo_ctrl.met_cool_down.gui_index_ln2_ctrl := 3; }
        RadioButton (134,0 33x103), variable: MAIN.met_cryo_ctrl.met_cool_down.gui_index_ln2_ctrl-1
            Areas[0]: Text=Radiobutton
            Areas[1]: Text=Radiobutton
END_VISUALIZATION

// HMI/VISUs/Subsystems/CRY/Components/VISU_HMI_CRY_RH
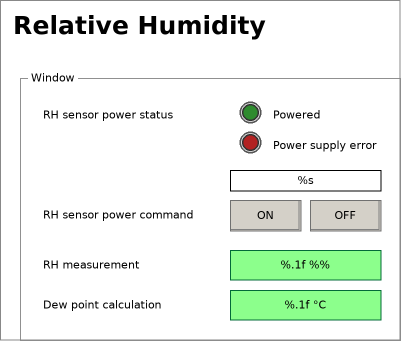
VISUALIZATION VISU_HMI_CRY_RH  // 401x341
VAR_IN_OUT
	m_Instance : FB_METIS_RH;
END_VAR
    Label (10,10 299x30), "Relative Humidity"
    GroupBox (20,70 381x271), "Window"
        Rectangle (210,180 151x30), "%.1f %%", text variable: m_Instance.rh_cry_wi.stat.lrRhPercent, colour toggle: NOT m_Instance.rh_cry_wi.stat.bValid
        Label (20,180 131x30), "RH measurement"
        Rectangle (210,220 151x30), "%.1f °C", text variable: m_Instance.rh_cry_wi.stat.lrDewPointTempC, colour toggle: NOT m_Instance.rh_cry_wi.stat.bDewPointTempValid
        Label (20,220 141x30), "Dew point calculation"
        Button (210,130 71x31), "ON", input disabled if: m_Instance.rh_cry_wi.power.stat.bActive
            OnMouseClick: execute { m_Instance.rh_cry_wi.power.ctrl.bEnable := TRUE; }
        Label (20,30 161x30), "RH sensor power status"
        Button (290,130 71x31), "OFF", input disabled if: NOT m_Instance.rh_cry_wi.power.stat.bActive
            OnMouseClick: execute { m_Instance.rh_cry_wi.power.ctrl.bEnable := FALSE; }
        Lamp1 (210,30 41x25), variable: m_Instance.rh_cry_wi.power.stat.bActive, style: Lamp-Lamp1-Green
        Label (250,30 61x30), "Powered"
        Label (250,60 121x31), "Power supply error"
        Rectangle (210,100 151x21), "%s", text variable: m_Instance.rh_cry_wi.power.stat.sStatus
        Label (20,130 171x30), "RH sensor power command"
    Lamp1 (230,130 41x25), variable: m_Instance.rh_cry_wi.power.stat.bError, style: Lamp-Lamp1-Red
END_VISUALIZATION

// HMI/VISUs/Subsystems/CRY/Components/VISU_HMI_CRY_TCTRL
